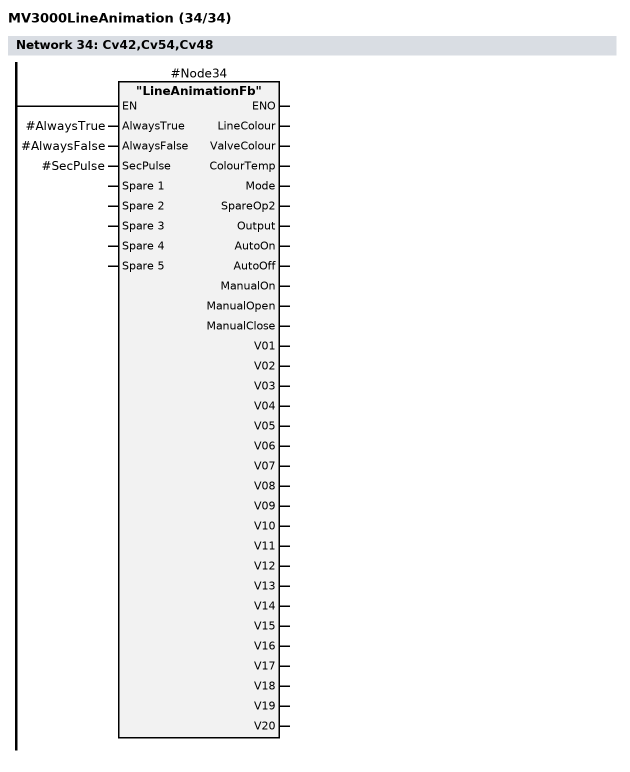
   RUNG wire#powerrail
      #Node34(AlwaysTrue := #AlwaysTrue, AlwaysFalse := #AlwaysFalse, SecPulse := #SecPulse, "Spare 1" :=, "Spare 2" :=, "Spare 3" :=, "Spare 4" :=, "Spare 5" :=, LineColour =>, ValveColour =>, ColourTemp =>, Mode =>, SpareOp2 =>, Output =>, AutoOn =>, AutoOff =>, ManualOn =>, ManualOpen =>, ManualClose =>, V01 =>, V02 =>, V03 =>, V04 =>, V05 =>, V06 =>, V07 =>, V08 =>, V09 =>, V10 =>, V11 =>, V12 =>, V13 =>, V14 =>, V15 =>, V16 =>, V17 =>, V18 =>, V19 =>, V20 =>)
   END_RUNG
   // the same network as SCL:
   #Node34(AlwaysTrue := #AlwaysTrue, AlwaysFalse := #AlwaysFalse, SecPulse := #SecPulse);   // "LineAnimationFb"
END_REGION
END_FUNCTION_BLOCK

FUNCTION_BLOCK "LineAnimationFb"   // FB802, LAD
{ S7_Optimized_Access := 'FALSE' }
// stored: AutoNumber false, SetENOAutomatically false
   VAR_INPUT
      AlwaysTrue : Bool;
      AlwaysFalse : Bool;
      SecPulse : Bool;
      "Spare 1" : Bool;
      "Spare 2" : Bool;
      "Spare 3" : Bool;
      "Spare 4" : Bool;
      "Spare 5" : Bool;
   END_VAR
   VAR_OUTPUT
      LineColour : DInt;
      ValveColour : DInt;
      ColourTemp : Int;
      Mode : Int;   // 0 - Force Close, 1- AutoOn, 2-ForceOn
      SpareOp2 : Int;
      Output : Bool;
      AutoOn : Bool;
      AutoOff : Bool;
      ManualOn : Bool;
      ManualOpen : Bool;
      ManualClose : Bool;
      V01 { ExternalAccessible := 'False'; ExternalVisible := 'False'; ExternalWritable := 'False'} : "LineAnimation";
      V02 { ExternalAccessible := 'False'; ExternalVisible := 'False'; ExternalWritable := 'False'} : "LineAnimation";
      V03 { ExternalAccessible := 'False'; ExternalVisible := 'False'; ExternalWritable := 'False'} : "LineAnimation";
      V04 { ExternalAccessible := 'False'; ExternalVisible := 'False'; ExternalWritable := 'False'} : "LineAnimation";
      V05 { ExternalAccessible := 'False'; ExternalVisible := 'False'; ExternalWritable := 'False'} : "LineAnimation";
      V06 { ExternalAccessible := 'False'; ExternalVisible := 'False'; ExternalWritable := 'False'} : "LineAnimation";
      V07 { ExternalAccessible := 'False'; ExternalVisible := 'False'; ExternalWritable := 'False'} : "LineAnimation";
      V08 { ExternalAccessible := 'False'; ExternalVisible := 'False'; ExternalWritable := 'False'} : "LineAnimation";
      V09 { ExternalAccessible := 'False'; ExternalVisible := 'False'; ExternalWritable := 'False'} : "LineAnimation";
      V10 { ExternalAccessible := 'False'; ExternalVisible := 'False'; ExternalWritable := 'False'} : "LineAnimation";
      V11 { ExternalAccessible := 'False'; ExternalVisible := 'False'; ExternalWritable := 'False'} : "LineAnimation";
      V12 { ExternalAccessible := 'False'; ExternalVisible := 'False'; ExternalWritable := 'False'} : "LineAnimation";
      V13 { ExternalAccessible := 'False'; ExternalVisible := 'False'; ExternalWritable := 'False'} : "LineAnimation";
      V14 { ExternalAccessible := 'False'; ExternalVisible := 'False'; ExternalWritable := 'False'} : "LineAnimation";
      V15 { ExternalAccessible := 'False'; ExternalVisible := 'False'; ExternalWritable := 'False'} : "LineAnimation";
      V16 { ExternalAccessible := 'False'; ExternalVisible := 'False'; ExternalWritable := 'False'} : "LineAnimation";
      V17 { ExternalAccessible := 'False'; ExternalVisible := 'False'; ExternalWritable := 'False'} : "LineAnimation";
      V18 { ExternalAccessible := 'False'; ExternalVisible := 'False'; ExternalWritable := 'False'} : "LineAnimation";
      V19 { ExternalAccessible := 'False'; ExternalVisible := 'False'; ExternalWritable := 'False'} : "LineAnimation";
      V20 { ExternalAccessible := 'False'; ExternalVisible := 'False'; ExternalWritable := 'False'} : "LineAnimation";
   END_VAR
BEGIN

REGION Network 1: Auto On
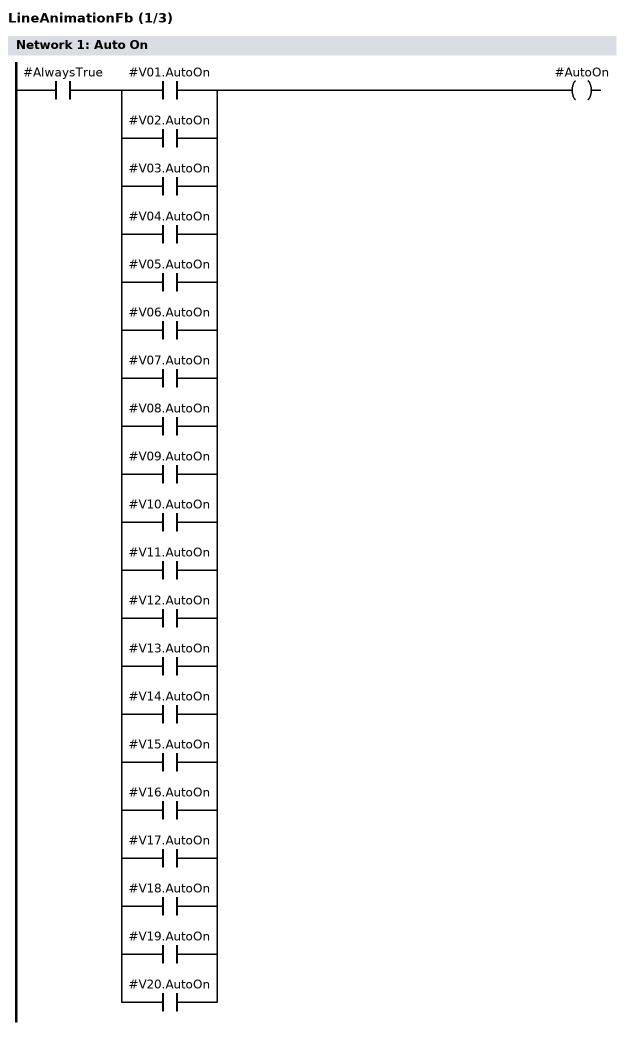
   RUNG wire#powerrail
      Contact( #AlwaysTrue )
      wire#w1
      Contact( #V01.AutoOn )
      wire#w2
      Coil( #AutoOn )
   END_RUNG
   RUNG wire#w1
      Contact( #V02.AutoOn )
   END_RUNG wire#w2
   RUNG wire#w1
      Contact( #V03.AutoOn )
   END_RUNG wire#w2
   RUNG wire#w1
      Contact( #V04.AutoOn )
   END_RUNG wire#w2
   RUNG wire#w1
      Contact( #V05.AutoOn )
   END_RUNG wire#w2
   RUNG wire#w1
      Contact( #V06.AutoOn )
   END_RUNG wire#w2
   RUNG wire#w1
      Contact( #V07.AutoOn )
   END_RUNG wire#w2
   RUNG wire#w1
      Contact( #V08.AutoOn )
   END_RUNG wire#w2
   RUNG wire#w1
      Contact( #V09.AutoOn )
   END_RUNG wire#w2
   RUNG wire#w1
      Contact( #V10.AutoOn )
   END_RUNG wire#w2
   RUNG wire#w1
      Contact( #V11.AutoOn )
   END_RUNG wire#w2
   RUNG wire#w1
      Contact( #V12.AutoOn )
   END_RUNG wire#w2
   RUNG wire#w1
      Contact( #V13.AutoOn )
   END_RUNG wire#w2
   RUNG wire#w1
      Contact( #V14.AutoOn )
   END_RUNG wire#w2
   RUNG wire#w1
      Contact( #V15.AutoOn )
   END_RUNG wire#w2
   RUNG wire#w1
      Contact( #V16.AutoOn )
   END_RUNG wire#w2
   RUNG wire#w1
      Contact( #V17.AutoOn )
   END_RUNG wire#w2
   RUNG wire#w1
      Contact( #V18.AutoOn )
   END_RUNG wire#w2
   RUNG wire#w1
      Contact( #V19.AutoOn )
   END_RUNG wire#w2
   RUNG wire#w1
      Contact( #V20.AutoOn )
   END_RUNG wire#w2
   // the same network as SCL:
   #AutoOn := #AlwaysTrue AND (#V01.AutoOn OR #V02.AutoOn OR #V03.AutoOn OR #V04.AutoOn OR #V05.AutoOn OR #V06.AutoOn OR #V07.AutoOn OR #V08.AutoOn OR #V09.AutoOn OR #V10.AutoOn OR #V11.AutoOn OR #V12.AutoOn OR #V13.AutoOn OR #V14.AutoOn OR #V15.AutoOn OR #V16.AutoOn OR #V17.AutoOn OR #V18.AutoOn OR #V19.AutoOn OR #V20.AutoOn);
END_REGION

REGION Network 2: Force Open
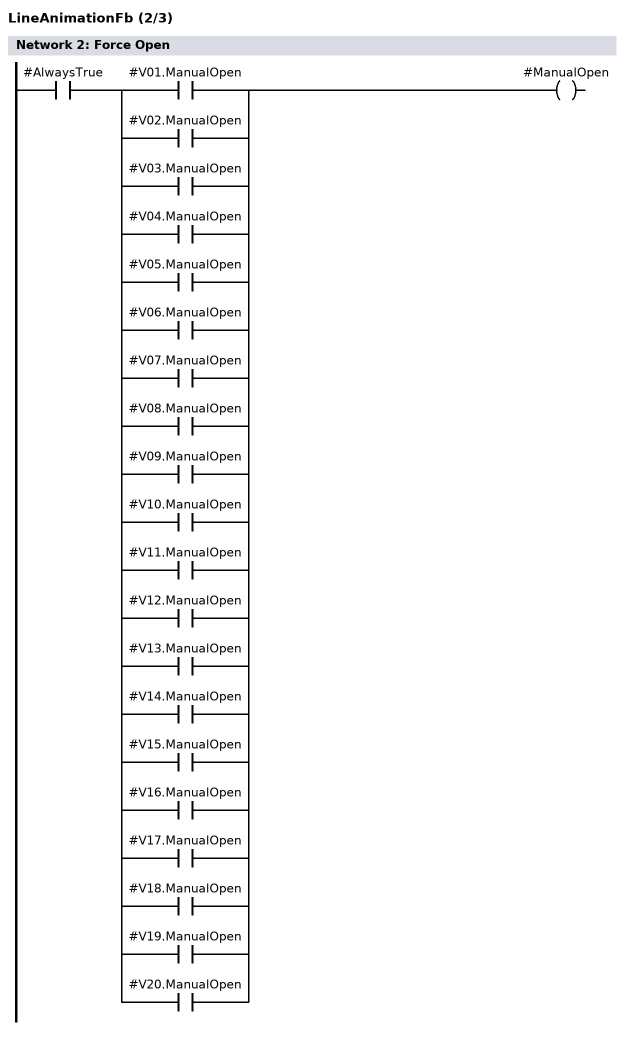
   RUNG wire#powerrail
      Contact( #AlwaysTrue )
      wire#w1
      Contact( #V01.ManualOpen )
      wire#w2
      Coil( #ManualOpen )
   END_RUNG
   RUNG wire#w1
      Contact( #V02.ManualOpen )
   END_RUNG wire#w2
   RUNG wire#w1
      Contact( #V03.ManualOpen )
   END_RUNG wire#w2
   RUNG wire#w1
      Contact( #V04.ManualOpen )
   END_RUNG wire#w2
   RUNG wire#w1
      Contact( #V05.ManualOpen )
   END_RUNG wire#w2
   RUNG wire#w1
      Contact( #V06.ManualOpen )
   END_RUNG wire#w2
   RUNG wire#w1
      Contact( #V07.ManualOpen )
   END_RUNG wire#w2
   RUNG wire#w1
      Contact( #V08.ManualOpen )
   END_RUNG wire#w2
   RUNG wire#w1
      Contact( #V09.ManualOpen )
   END_RUNG wire#w2
   RUNG wire#w1
      Contact( #V10.ManualOpen )
   END_RUNG wire#w2
   RUNG wire#w1
      Contact( #V11.ManualOpen )
   END_RUNG wire#w2
   RUNG wire#w1
      Contact( #V12.ManualOpen )
   END_RUNG wire#w2
   RUNG wire#w1
      Contact( #V13.ManualOpen )
   END_RUNG wire#w2
   RUNG wire#w1
      Contact( #V14.ManualOpen )
   END_RUNG wire#w2
   RUNG wire#w1
      Contact( #V15.ManualOpen )
   END_RUNG wire#w2
   RUNG wire#w1
      Contact( #V16.ManualOpen )
   END_RUNG wire#w2
   RUNG wire#w1
      Contact( #V17.ManualOpen )
   END_RUNG wire#w2
   RUNG wire#w1
      Contact( #V18.ManualOpen )
   END_RUNG wire#w2
   RUNG wire#w1
      Contact( #V19.ManualOpen )
   END_RUNG wire#w2
   RUNG wire#w1
      Contact( #V20.ManualOpen )
   END_RUNG wire#w2
   // the same network as SCL:
   #ManualOpen := #AlwaysTrue AND (#V01.ManualOpen OR #V02.ManualOpen OR #V03.ManualOpen OR #V04.ManualOpen OR #V05.ManualOpen OR #V06.ManualOpen OR #V07.ManualOpen OR #V08.ManualOpen OR #V09.ManualOpen OR #V10.ManualOpen OR #V11.ManualOpen OR #V12.ManualOpen OR #V13.ManualOpen OR #V14.ManualOpen OR #V15.ManualOpen OR #V16.ManualOpen OR #V17.ManualOpen OR #V18.ManualOpen OR #V19.ManualOpen OR #V20.ManualOpen);
END_REGION

REGION Network 3: Line Colour
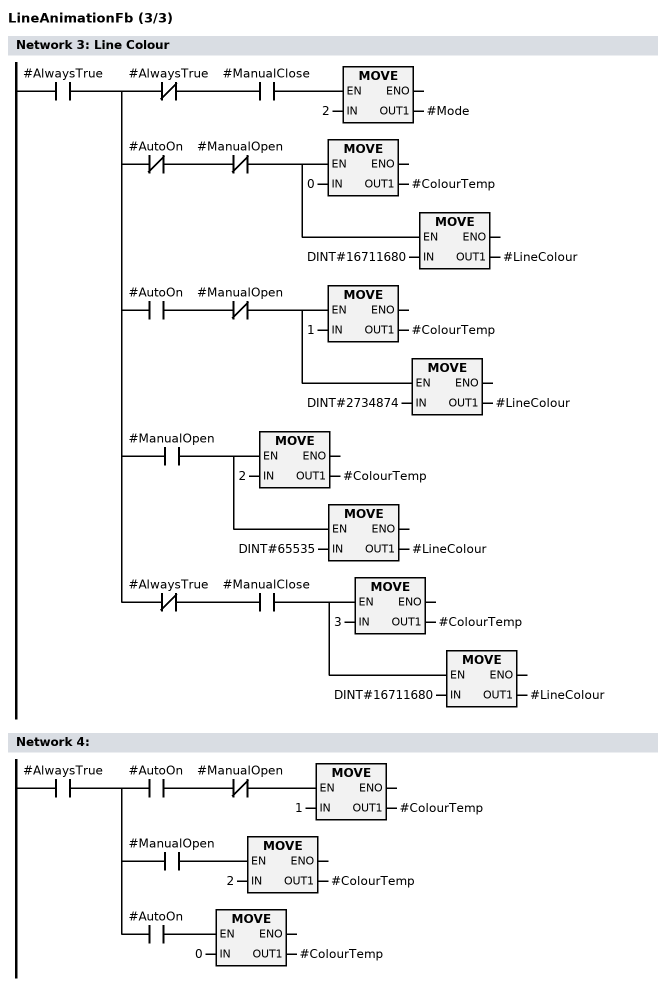
   RUNG wire#powerrail
      Contact( #AlwaysTrue )
      wire#w1
      I_Contact( #AlwaysTrue )
      Contact( #ManualClose )
      Move(in := 2, out1 => #Mode)
   END_RUNG
   RUNG wire#w1
      I_Contact( #AutoOn )
      I_Contact( #ManualOpen )
      wire#w2
      Move(in := 0, out1 => #ColourTemp)
   END_RUNG
   RUNG wire#w2
      Move(in := DINT#16711680, out1 => #LineColour)
   END_RUNG
   RUNG wire#w1
      Contact( #AutoOn )
      I_Contact( #ManualOpen )
      wire#w3
      Move(in := 1, out1 => #ColourTemp)
   END_RUNG
   RUNG wire#w3
      Move(in := DINT#2734874, out1 => #LineColour)
   END_RUNG
   RUNG wire#w1
      Contact( #ManualOpen )
      wire#w4
      Move(in := 2, out1 => #ColourTemp)
   END_RUNG
   RUNG wire#w4
      Move(in := DINT#65535, out1 => #LineColour)
   END_RUNG
   RUNG wire#w1
      I_Contact( #AlwaysTrue )
      Contact( #ManualClose )
      wire#w5
      Move(in := 3, out1 => #ColourTemp)
   END_RUNG
   RUNG wire#w5
      Move(in := DINT#16711680, out1 => #LineColour)
   END_RUNG
   // the same network as SCL:
   IF #AlwaysTrue AND NOT #AlwaysTrue AND #ManualClose THEN #Mode := 2; END_IF;
   IF #AlwaysTrue AND NOT #AutoOn AND NOT #ManualOpen THEN
       #ColourTemp := 0;
       #LineColour := DINT#16711680;
   END_IF;
   IF #AlwaysTrue AND #AutoOn AND NOT #ManualOpen THEN
       #ColourTemp := 1;
       #LineColour := DINT#2734874;
   END_IF;
   IF #AlwaysTrue AND #ManualOpen THEN
       #ColourTemp := 2;
       #LineColour := DINT#65535;
   END_IF;
   IF #AlwaysTrue AND NOT #AlwaysTrue AND #ManualClose THEN
       #ColourTemp := 3;
       #LineColour := DINT#16711680;
   END_IF;
END_REGION

REGION Network 4
   RUNG wire#powerrail
      Contact( #AlwaysTrue )
      wire#w1
      Contact( #AutoOn )
      I_Contact( #ManualOpen )
      Move(in := 1, out1 => #ColourTemp)
   END_RUNG
   RUNG wire#w1
      Contact( #ManualOpen )
      Move(in := 2, out1 => #ColourTemp)
   END_RUNG
   RUNG wire#w1
      Contact( #AutoOn )
      Move(in := 0, out1 => #ColourTemp)
   END_RUNG
   // the same network as SCL:
   IF #AlwaysTrue AND #AutoOn AND NOT #ManualOpen THEN #ColourTemp := 1; END_IF;
   IF #AlwaysTrue AND #ManualOpen THEN #ColourTemp := 2; END_IF;
   IF #AlwaysTrue AND #AutoOn THEN #ColourTemp := 0; END_IF;
END_REGION
END_FUNCTION_BLOCK

FUNCTION "MV3000LineAnimationFc" : Void
{ S7_Optimized_Access := 'FALSE' }
VERSION : 0.1

BEGIN
	//////////////////////////////////// AUTO ON ////////////////////////////////////////////
	//AutoON
	"MV3000LineAnimationDb"."Node 1".V01.AutoOn := "ValvesOutputDb".Cv01;
	"MV3000LineAnimationDb"."Node 1".V02.AutoOn := "ValvesOutputDb".Cv02;
	"MV3000LineAnimationDb"."Node 1".V03.AutoOn := "ValvesOutputDb".Cv10;
	
	
	"MV3000LineAnimationDb"."Node 2".V01.AutoOn := "ValvesOutputDb".Cv03;
	"MV3000LineAnimationDb"."Node 2".V02.AutoOn := "ValvesOutputDb".Cv04;
	"MV3000LineAnimationDb"."Node 2".V03.AutoOn := "ValvesOutputDb".Cv05;
	"MV3000LineAnimationDb"."Node 2".V04.AutoOn := "ValvesOutputDb".Cv06;
	
	
	"MV3000LineAnimationDb"."Node 3".V01.AutoOn := "ValvesOutputDb".Cv07;
	"MV3000LineAnimationDb"."Node 3".V02.AutoOn := "ValvesOutputDb".Cv08;
	"MV3000LineAnimationDb"."Node 3".V03.AutoOn := "ValvesOutputDb".Cv09;
	
	
	"MV3000LineAnimationDb"."Node 4".V01.AutoOn := "ValvesOutputDb".Cv16;
	"MV3000LineAnimationDb"."Node 4".V02.AutoOn := "ValvesOutputDb".Cv17;
	"MV3000LineAnimationDb"."Node 4".V03.AutoOn := "ValvesOutputDb".Cv22;
	"MV3000LineAnimationDb"."Node 4".V04.AutoOn := "ValvesOutputDb".Cv23;
	"MV3000LineAnimationDb"."Node 4".V05.AutoOn := "ValvesOutputDb".Cv24;
	"MV3000LineAnimationDb"."Node 4".V06.AutoOn := "ValvesOutputDb".Cv25;
	
	
	"MV3000LineAnimationDb"."Node 5".V01.AutoOn := "ValvesOutputDb".Cv22;
	"MV3000LineAnimationDb"."Node 5".V02.AutoOn := "ValvesOutputDb".Cv25;
	
	
	"MV3000LineAnimationDb"."Node 6".V01.AutoOn := "ValvesOutputDb".Cv18;
	"MV3000LineAnimationDb"."Node 6".V02.AutoOn := "ValvesOutputDb".Cv19;
	"MV3000LineAnimationDb"."Node 6".V03.AutoOn := "ValvesOutputDb".Cv20;
	"MV3000LineAnimationDb"."Node 6".V04.AutoOn := "ValvesOutputDb".Cv21;
	
	"MV3000LineAnimationDb"."Node 7".V01.AutoOn := "ValvesOutputDb".Cv19;
	"MV3000LineAnimationDb"."Node 7".V02.AutoOn := "ValvesOutputDb".Cv20;
	
	"MV3000LineAnimationDb"."Node 8".V01.AutoOn := "ValvesOutputDb".Cv16;
	"MV3000LineAnimationDb"."Node 8".V02.AutoOn := "ValvesOutputDb".Cv15;
	"MV3000LineAnimationDb"."Node 8".V03.AutoOn := "ValvesOutputDb".Cv63;
	
	"MV3000LineAnimationDb"."Node 9".V01.AutoOn := "ValvesOutputDb".Cv10;
	"MV3000LineAnimationDb"."Node 9".V02.AutoOn := "ValvesOutputDb".Cv11;
	"MV3000LineAnimationDb"."Node 9".V03.AutoOn := "ValvesOutputDb".Cv12;
	"MV3000LineAnimationDb"."Node 9".V04.AutoOn := "ValvesOutputDb".Cv13;
	"MV3000LineAnimationDb"."Node 9".V05.AutoOn := "ValvesOutputDb".Cv14;
	"MV3000LineAnimationDb"."Node 9".V06.AutoOn := "ValvesOutputDb".Cv15;
	
	"MV3000LineAnimationDb"."Node 10".V01.AutoOn := "ValvesOutputDb".Cv11;
	"MV3000LineAnimationDb"."Node 10".V02.AutoOn := "ValvesOutputDb".Cv39;
	
	"MV3000LineAnimationDb"."Node 11".V01.AutoOn := "ValvesOutputDb".Cv12;
	"MV3000LineAnimationDb"."Node 11".V02.AutoOn := "ValvesOutputDb".Cv26;
	"MV3000LineAnimationDb"."Node 11".V03.AutoOn := "ValvesOutputDb".Cv64;
	
	"MV3000LineAnimationDb"."Node 12".V01.AutoOn := "ValvesOutputDb".Cv31;
	"MV3000LineAnimationDb"."Node 12".V02.AutoOn := "ValvesOutputDb".Cv41;
	
	"MV3000LineAnimationDb"."Node 13".V01.AutoOn := "ValvesOutputDb".Fbov01;
	"MV3000LineAnimationDb"."Node 13".V02.AutoOn := "ValvesOutputDb".Cv30;
	"MV3000LineAnimationDb"."Node 13".V03.AutoOn := "ValvesOutputDb".Cv31;
	"MV3000LineAnimationDb"."Node 13".V04.AutoOn := "ValvesOutputDb".Cv32;
	"MV3000LineAnimationDb"."Node 13".V05.AutoOn := "ValvesOutputDb".Cv33;
	
	"MV3000LineAnimationDb"."Node 14".V01.AutoOn := "ValvesOutputDb".Cv27;
	"MV3000LineAnimationDb"."Node 14".V02.AutoOn := "ValvesOutputDb".Cv28;
	"MV3000LineAnimationDb"."Node 14".V03.AutoOn := "ValvesOutputDb".Cv29;
	
	"MV3000LineAnimationDb"."Node 15".V01.AutoOn := "ValvesOutputDb".Cv30;
	"MV3000LineAnimationDb"."Node 15".V02.AutoOn := "ValvesOutputDb".Cv33;
	"MV3000LineAnimationDb"."Node 15".V03.AutoOn := "ValvesOutputDb".Cv34;
	"MV3000LineAnimationDb"."Node 15".V04.AutoOn := "ValvesOutputDb".Cv35;
	
	"MV3000LineAnimationDb"."Node 16".V01.AutoOn := "ValvesOutputDb".Cv32;
	"MV3000LineAnimationDb"."Node 16".V02.AutoOn := "ValvesOutputDb".Cv36;
	"MV3000LineAnimationDb"."Node 16".V03.AutoOn := "ValvesOutputDb".Cv39;
	"MV3000LineAnimationDb"."Node 16".V04.AutoOn := "ValvesOutputDb".Cv40;
	
	"MV3000LineAnimationDb"."Node 17".V01.AutoOn := "ValvesOutputDb".Cv40;
	"MV3000LineAnimationDb"."Node 17".V02.AutoOn := "ValvesOutputDb".Cv41;
	"MV3000LineAnimationDb"."Node 17".V03.AutoOn := "ValvesOutputDb".Cv42;
	"MV3000LineAnimationDb"."Node 17".V04.AutoOn := "ValvesOutputDb".Cv43;
	"MV3000LineAnimationDb"."Node 17".V05.AutoOn := "ValvesOutputDb".Cv44;
	
	"MV3000LineAnimationDb"."Node 18".V01.AutoOn := "ValvesOutputDb".Cv43;
	"MV3000LineAnimationDb"."Node 18".V02.AutoOn := "ValvesOutputDb".Cv47;
	"MV3000LineAnimationDb"."Node 18".V03.AutoOn := "ValvesOutputDb".Cv48;
	"MV3000LineAnimationDb"."Node 18".V04.AutoOn := "ValvesOutputDb".Cv49;
	"MV3000LineAnimationDb"."Node 18".V05.AutoOn := "ValvesOutputDb".Cv50;
	
	
	"MV3000LineAnimationDb"."Node 19".V01.AutoOn := "ValvesOutputDb".Cv49;
	"MV3000LineAnimationDb"."Node 19".V02.AutoOn := "ValvesOutputDb".Cv53;
	"MV3000LineAnimationDb"."Node 19".V03.AutoOn := "ValvesOutputDb".Cv54;
	"MV3000LineAnimationDb"."Node 19".V04.AutoOn := "ValvesOutputDb".Cv55;
	"MV3000LineAnimationDb"."Node 19".V05.AutoOn := "ValvesOutputDb".Cv56;
	
	"MV3000LineAnimationDb"."Node 20".V01.AutoOn := "ValvesOutputDb".Cv55;
	"MV3000LineAnimationDb"."Node 20".V02.AutoOn := "ValvesOutputDb".Cv61;
	"MV3000LineAnimationDb"."Node 20".V03.AutoOn := "ValvesOutputDb".Cv62;
	
	
	"MV3000LineAnimationDb"."Node 21".V01.AutoOn := "ValvesOutputDb".Cv59;
	"MV3000LineAnimationDb"."Node 21".V02.AutoOn := "ValvesOutputDb".Cv60;
	"MV3000LineAnimationDb"."Node 21".V03.AutoOn := "ValvesOutputDb".Cv61;
	
	"MV3000LineAnimationDb"."Node 22".V01.AutoOn := "ValvesOutputDb".Cv56;
	"MV3000LineAnimationDb"."Node 22".V02.AutoOn := "ValvesOutputDb".Cv58;
	"MV3000LineAnimationDb"."Node 22".V03.AutoOn := "ValvesOutputDb".Cv57;
	
	"MV3000LineAnimationDb"."Node 23".V01.AutoOn := "ValvesOutputDb".Cv50;
	"MV3000LineAnimationDb"."Node 23".V02.AutoOn := "ValvesOutputDb".Cv51;
	"MV3000LineAnimationDb"."Node 23".V03.AutoOn := "ValvesOutputDb".Cv52;
	"MV3000LineAnimationDb"."Node 23".V04.AutoOn := "ValvesOutputDb".Cv53;
	
	
	"MV3000LineAnimationDb"."Node 24".V01.AutoOn := "ValvesOutputDb".Cv44;
	"MV3000LineAnimationDb"."Node 24".V02.AutoOn := "ValvesOutputDb".Cv45;
	"MV3000LineAnimationDb"."Node 24".V03.AutoOn := "ValvesOutputDb".Cv46;
	"MV3000LineAnimationDb"."Node 24".V04.AutoOn := "ValvesOutputDb".Cv47;
	
	"MV3000LineAnimationDb"."Node 25".V01.AutoOn := "ValvesOutputDb".Cv36;
	"MV3000LineAnimationDb"."Node 25".V02.AutoOn := "ValvesOutputDb".Cv37;
	"MV3000LineAnimationDb"."Node 25".V03.AutoOn := "ValvesOutputDb".Cv38;
	
	
	"MV3000LineAnimationDb"."Node 26".V01.AutoOn := "ValvesOutputDb".Cv30;
	"MV3000LineAnimationDb"."Node 26".V02.AutoOn := "ValvesOutputDb".Cv33;
	"MV3000LineAnimationDb"."Node 26".V03.AutoOn := "ValvesOutputDb".Cv34;
	"MV3000LineAnimationDb"."Node 26".V04.AutoOn := "ValvesOutputDb".Cv35;
	
	"MV3000LineAnimationDb"."Node 27".V01.AutoOn := "ValvesOutputDb".Cv28;
	"MV3000LineAnimationDb"."Node 27".V02.AutoOn := "ValvesOutputDb".Cv34;
	"MV3000LineAnimationDb"."Node 27".V03.AutoOn := "ValvesOutputDb".Cv37;
	"MV3000LineAnimationDb"."Node 27".V04.AutoOn := "ValvesOutputDb".Cv45;
	"MV3000LineAnimationDb"."Node 27".V05.AutoOn := "ValvesOutputDb".Cv51;
	"MV3000LineAnimationDb"."Node 27".V06.AutoOn := "ValvesOutputDb".Cv57;
	"MV3000LineAnimationDb"."Node 27".V07.AutoOn := "ValvesOutputDb".Cv60;
	
	"MV3000LineAnimationDb"."Node 28".V01.AutoOn := "ValvesOutputDb".Cv22;
	"MV3000LineAnimationDb"."Node 28".V02.AutoOn := "ValvesOutputDb".Cv19;
	"MV3000LineAnimationDb"."Node 28".V03.AutoOn := "ValvesOutputDb".Cv25;
	"MV3000LineAnimationDb"."Node 28".V04.AutoOn := "ValvesOutputDb".Cv20;
	"MV3000LineAnimationDb"."Node 28".V05.AutoOn := "ValvesOutputDb".Cv29;
	"MV3000LineAnimationDb"."Node 28".V06.AutoOn := "ValvesOutputDb".Cv35;
	"MV3000LineAnimationDb"."Node 28".V07.AutoOn := "ValvesOutputDb".Cv38;
	"MV3000LineAnimationDb"."Node 28".V08.AutoOn := "ValvesOutputDb".Cv46;
	"MV3000LineAnimationDb"."Node 28".V09.AutoOn := "ValvesOutputDb".Cv52;
	"MV3000LineAnimationDb"."Node 28".V10.AutoOn := "ValvesOutputDb".Cv58;
	"MV3000LineAnimationDb"."Node 28".V11.AutoOn := "ValvesOutputDb".Cv59;
	
	"MV3000LineAnimationDb"."Node 29".V01.AutoOn := "ValvesOutputDb".Cv04;
	"MV3000LineAnimationDb"."Node 29".V02.AutoOn := "ValvesOutputDb".Cv01;
	
	"MV3000LineAnimationDb"."Node 30".V01.AutoOn := "ValvesOutputDb".Cv06;
	"MV3000LineAnimationDb"."Node 30".V02.AutoOn := "ValvesOutputDb".Cv09;
	
	"MV3000LineAnimationDb"."Node31".V01.AutoOn :="ValvesOutputDb".Cv06;
	"MV3000LineAnimationDb"."Node31".V02.AutoOn := "ValvesOutputDb".Cv09;
	"MV3000LineAnimationDb"."Node31".V03.AutoOn := "ValvesOutputDb".Cv08;
	
	"MV3000LineAnimationDb".Node32.V01.AutoOn := "ValvesOutputDb".Cv05;
	"MV3000LineAnimationDb".Node32.V02.AutoOn := "ValvesOutputDb".Cv24;
	
	"MV3000LineAnimationDb".Node33.V01.AutoOn := "ValvesOutputDb".Fbov01;
	"MV3000LineAnimationDb".Node33.V02.AutoOn := "ValvesOutputDb".Cv26;
	
	
	"MV3000LineAnimationDb".Node34.V01.AutoOn := "ValvesOutputDb".Cv42;
	"MV3000LineAnimationDb".Node34.V02.AutoOn := "ValvesOutputDb".Cv54;
	"MV3000LineAnimationDb".Node34.V03.AutoOn := "ValvesOutputDb".Cv48;
	
	
	
	
	
	//////////////////////////////////////////  MANUAL OPEN /////////////////////////////////////////////
	
	//ManualOpen
	
	"MV3000LineAnimationDb"."Node 1".V01.ManualOpen := "DO_FaceplateDb".Cv01.ValveOpen;
	"MV3000LineAnimationDb"."Node 1".V02.ManualOpen := "DO_FaceplateDb".Cv02.ValveOpen;
	"MV3000LineAnimationDb"."Node 1".V03.ManualOpen := "DO_FaceplateDb".Cv10.ValveOpen;
	
	
	"MV3000LineAnimationDb"."Node 2".V01.ManualOpen := "DO_FaceplateDb".Cv03.ValveOpen;
	"MV3000LineAnimationDb"."Node 2".V02.ManualOpen := "DO_FaceplateDb".Cv04.ValveOpen;
	"MV3000LineAnimationDb"."Node 2".V03.ManualOpen := "DO_FaceplateDb".Cv05.ValveOpen;
	"MV3000LineAnimationDb"."Node 2".V04.ManualOpen := "DO_FaceplateDb".Cv06.ValveOpen;
	
	
	"MV3000LineAnimationDb"."Node 3".V01.ManualOpen := "DO_FaceplateDb".Cv07.ValveOpen;
	"MV3000LineAnimationDb"."Node 3".V02.ManualOpen := "DO_FaceplateDb".Cv08.ValveOpen;
	"MV3000LineAnimationDb"."Node 3".V03.ManualOpen := "DO_FaceplateDb".Cv09.ValveOpen;
	
	
	"MV3000LineAnimationDb"."Node 4".V01.ManualOpen := "DO_FaceplateDb".Cv16.ValveOpen;
	"MV3000LineAnimationDb"."Node 4".V02.ManualOpen := "DO_FaceplateDb".Cv17.ValveOpen;
	"MV3000LineAnimationDb"."Node 4".V03.ManualOpen := "DO_FaceplateDb".Cv22.ValveOpen;
	"MV3000LineAnimationDb"."Node 4".V04.ManualOpen := "DO_FaceplateDb".Cv23.ValveOpen;
	"MV3000LineAnimationDb"."Node 4".V05.ManualOpen := "DO_FaceplateDb".Cv24.ValveOpen;
	"MV3000LineAnimationDb"."Node 4".V06.ManualOpen := "DO_FaceplateDb".Cv25.ValveOpen;
	
	
	"MV3000LineAnimationDb"."Node 5".V01.ManualOpen := "DO_FaceplateDb".Cv22.ValveOpen;
	"MV3000LineAnimationDb"."Node 5".V02.ManualOpen := "DO_FaceplateDb".Cv25.ValveOpen;
	
	
	"MV3000LineAnimationDb"."Node 6".V01.ManualOpen := "DO_FaceplateDb".Cv18.ValveOpen;
	"MV3000LineAnimationDb"."Node 6".V02.ManualOpen := "DO_FaceplateDb".Cv19.ValveOpen;
	"MV3000LineAnimationDb"."Node 6".V03.ManualOpen := "DO_FaceplateDb".Cv20.ValveOpen;
	"MV3000LineAnimationDb"."Node 6".V04.ManualOpen := "DO_FaceplateDb".Cv21.ValveOpen;
	
	"MV3000LineAnimationDb"."Node 7".V01.ManualOpen := "DO_FaceplateDb".Cv19.ValveOpen;
	"MV3000LineAnimationDb"."Node 7".V02.ManualOpen := "DO_FaceplateDb".Cv20.ValveOpen;
	
	"MV3000LineAnimationDb"."Node 8".V01.ManualOpen := "DO_FaceplateDb".Cv16.ValveOpen;
	"MV3000LineAnimationDb"."Node 8".V02.ManualOpen := "DO_FaceplateDb".Cv15.ValveOpen;
	"MV3000LineAnimationDb"."Node 8".V03.ManualOpen := "DO_FaceplateDb".Cv63.ValveOpen;
	
	"MV3000LineAnimationDb"."Node 9".V01.ManualOpen := "DO_FaceplateDb".Cv10.ValveOpen;
	"MV3000LineAnimationDb"."Node 9".V02.ManualOpen := "DO_FaceplateDb".Cv11.ValveOpen;
	"MV3000LineAnimationDb"."Node 9".V03.ManualOpen := "DO_FaceplateDb".Cv12.ValveOpen;
	"MV3000LineAnimationDb"."Node 9".V04.ManualOpen := "DO_FaceplateDb".Cv13.ValveOpen;
	"MV3000LineAnimationDb"."Node 9".V05.ManualOpen := "DO_FaceplateDb".Cv14.ValveOpen;
	"MV3000LineAnimationDb"."Node 9".V06.ManualOpen := "DO_FaceplateDb".Cv15.ValveOpen;
	
	"MV3000LineAnimationDb"."Node 10".V01.ManualOpen := "DO_FaceplateDb".Cv11.ValveOpen;
	"MV3000LineAnimationDb"."Node 10".V02.ManualOpen := "DO_FaceplateDb".Cv39.ValveOpen;
	
	"MV3000LineAnimationDb"."Node 11".V01.ManualOpen := "DO_FaceplateDb".Cv12.ValveOpen;
	"MV3000LineAnimationDb"."Node 11".V02.ManualOpen := "DO_FaceplateDb".Cv26.ValveOpen;
	"MV3000LineAnimationDb"."Node 11".V03.ManualOpen := "DO_FaceplateDb".Cv64.ValveOpen;
	
	"MV3000LineAnimationDb"."Node 12".V01.ManualOpen := "DO_FaceplateDb".Cv31.ValveOpen;
	"MV3000LineAnimationDb"."Node 12".V02.ManualOpen := "DO_FaceplateDb".Cv41.ValveOpen;
	
	"MV3000LineAnimationDb"."Node 13".V01.ManualOpen := "DO_FaceplateDb".Fbov01.ValveOpen;
	"MV3000LineAnimationDb"."Node 13".V02.ManualOpen := "DO_FaceplateDb".Cv30.ValveOpen;
	"MV3000LineAnimationDb"."Node 13".V03.ManualOpen := "DO_FaceplateDb".Cv31.ValveOpen;
	"MV3000LineAnimationDb"."Node 13".V04.ManualOpen := "DO_FaceplateDb".Cv32.ValveOpen;
	"MV3000LineAnimationDb"."Node 13".V05.ManualOpen := "DO_FaceplateDb".Cv33.ValveOpen;
	
	"MV3000LineAnimationDb"."Node 14".V01.ManualOpen := "DO_FaceplateDb".Cv27.ValveOpen;
	"MV3000LineAnimationDb"."Node 14".V02.ManualOpen := "DO_FaceplateDb".Cv28.ValveOpen;
	"MV3000LineAnimationDb"."Node 14".V03.ManualOpen := "DO_FaceplateDb".Cv29.ValveOpen;
	
	"MV3000LineAnimationDb"."Node 15".V01.ManualOpen := "DO_FaceplateDb".Cv30.ValveOpen;
	"MV3000LineAnimationDb"."Node 15".V02.ManualOpen := "DO_FaceplateDb".Cv33.ValveOpen;
	"MV3000LineAnimationDb"."Node 15".V03.ManualOpen := "DO_FaceplateDb".Cv34.ValveOpen;
	"MV3000LineAnimationDb"."Node 15".V04.ManualOpen := "DO_FaceplateDb".Cv35.ValveOpen;
	
	"MV3000LineAnimationDb"."Node 16".V01.ManualOpen := "DO_FaceplateDb".Cv32.ValveOpen;
	"MV3000LineAnimationDb"."Node 16".V02.ManualOpen := "DO_FaceplateDb".Cv36.ValveOpen;
	"MV3000LineAnimationDb"."Node 16".V03.ManualOpen := "DO_FaceplateDb".Cv39.ValveOpen;
	"MV3000LineAnimationDb"."Node 16".V04.ManualOpen := "DO_FaceplateDb".Cv40.ValveOpen;
	
	"MV3000LineAnimationDb"."Node 17".V01.ManualOpen := "DO_FaceplateDb".Cv40.ValveOpen;
	"MV3000LineAnimationDb"."Node 17".V02.ManualOpen := "DO_FaceplateDb".Cv41.ValveOpen;
	"MV3000LineAnimationDb"."Node 17".V03.ManualOpen := "DO_FaceplateDb".Cv42.ValveOpen;
	"MV3000LineAnimationDb"."Node 17".V04.ManualOpen := "DO_FaceplateDb".Cv43.ValveOpen;
	"MV3000LineAnimationDb"."Node 17".V05.ManualOpen := "DO_FaceplateDb".Cv44.ValveOpen;
	
	"MV3000LineAnimationDb"."Node 18".V01.ManualOpen := "DO_FaceplateDb".Cv43.ValveOpen;
	"MV3000LineAnimationDb"."Node 18".V02.ManualOpen := "DO_FaceplateDb".Cv47.ValveOpen;
	"MV3000LineAnimationDb"."Node 18".V03.ManualOpen := "DO_FaceplateDb".Cv48.ValveOpen;
	"MV3000LineAnimationDb"."Node 18".V04.ManualOpen := "DO_FaceplateDb".Cv49.ValveOpen;
	"MV3000LineAnimationDb"."Node 18".V05.ManualOpen := "DO_FaceplateDb".Cv50.ValveOpen;
	
	
	"MV3000LineAnimationDb"."Node 19".V01.ManualOpen := "DO_FaceplateDb".Cv49.ValveOpen;
	"MV3000LineAnimationDb"."Node 19".V02.ManualOpen := "DO_FaceplateDb".Cv53.ValveOpen;
	"MV3000LineAnimationDb"."Node 19".V03.ManualOpen := "DO_FaceplateDb".Cv54.ValveOpen;
	"MV3000LineAnimationDb"."Node 19".V04.ManualOpen := "DO_FaceplateDb".Cv55.ValveOpen;
	"MV3000LineAnimationDb"."Node 19".V05.ManualOpen := "DO_FaceplateDb".Cv56.ValveOpen;
	
	"MV3000LineAnimationDb"."Node 20".V01.ManualOpen := "DO_FaceplateDb".Cv55.ValveOpen;
	"MV3000LineAnimationDb"."Node 20".V02.ManualOpen := "DO_FaceplateDb".Cv61.ValveOpen;
	"MV3000LineAnimationDb"."Node 20".V03.ManualOpen := "DO_FaceplateDb".Cv62.ValveOpen;
	
	
	"MV3000LineAnimationDb"."Node 21".V01.ManualOpen := "DO_FaceplateDb".Cv59.ValveOpen;
	"MV3000LineAnimationDb"."Node 21".V02.ManualOpen := "DO_FaceplateDb".Cv60.ValveOpen;
	"MV3000LineAnimationDb"."Node 21".V03.ManualOpen := "DO_FaceplateDb".Cv61.ValveOpen;
	
	"MV3000LineAnimationDb"."Node 22".V01.ManualOpen := "DO_FaceplateDb".Cv56.ValveOpen;
	"MV3000LineAnimationDb"."Node 22".V02.ManualOpen := "DO_FaceplateDb".Cv58.ValveOpen;
	"MV3000LineAnimationDb"."Node 22".V03.ManualOpen := "DO_FaceplateDb".Cv57.ValveOpen;
	
	"MV3000LineAnimationDb"."Node 23".V01.ManualOpen := "DO_FaceplateDb".Cv50.ValveOpen;
	"MV3000LineAnimationDb"."Node 23".V02.ManualOpen := "DO_FaceplateDb".Cv51.ValveOpen;
	"MV3000LineAnimationDb"."Node 23".V03.ManualOpen := "DO_FaceplateDb".Cv52.ValveOpen;
	"MV3000LineAnimationDb"."Node 23".V04.ManualOpen := "DO_FaceplateDb".Cv53.ValveOpen;
	
	
	"MV3000LineAnimationDb"."Node 24".V01.ManualOpen := "DO_FaceplateDb".Cv44.ValveOpen;
	"MV3000LineAnimationDb"."Node 24".V02.ManualOpen := "DO_FaceplateDb".Cv45.ValveOpen;
	"MV3000LineAnimationDb"."Node 24".V03.ManualOpen := "DO_FaceplateDb".Cv46.ValveOpen;
	"MV3000LineAnimationDb"."Node 24".V04.ManualOpen := "DO_FaceplateDb".Cv47.ValveOpen;
	
	"MV3000LineAnimationDb"."Node 25".V01.ManualOpen := "DO_FaceplateDb".Cv36.ValveOpen;
	"MV3000LineAnimationDb"."Node 25".V02.ManualOpen := "DO_FaceplateDb".Cv37.ValveOpen;
	"MV3000LineAnimationDb"."Node 25".V03.ManualOpen := "DO_FaceplateDb".Cv38.ValveOpen;
	
	
	"MV3000LineAnimationDb"."Node 26".V01.ManualOpen := "DO_FaceplateDb".Cv30.ValveOpen;
	"MV3000LineAnimationDb"."Node 26".V02.ManualOpen := "DO_FaceplateDb".Cv33.ValveOpen;
	"MV3000LineAnimationDb"."Node 26".V03.ManualOpen := "DO_FaceplateDb".Cv34.ValveOpen;
	"MV3000LineAnimationDb"."Node 26".V04.ManualOpen := "DO_FaceplateDb".Cv35.ValveOpen;
	
	"MV3000LineAnimationDb"."Node 27".V01.ManualOpen := "DO_FaceplateDb".Cv28.ValveOpen;
	"MV3000LineAnimationDb"."Node 27".V02.ManualOpen := "DO_FaceplateDb".Cv34.ValveOpen;
	"MV3000LineAnimationDb"."Node 27".V03.ManualOpen := "DO_FaceplateDb".Cv37.ValveOpen;
	"MV3000LineAnimationDb"."Node 27".V04.ManualOpen := "DO_FaceplateDb".Cv45.ValveOpen;
	"MV3000LineAnimationDb"."Node 27".V05.ManualOpen := "DO_FaceplateDb".Cv51.ValveOpen;
	"MV3000LineAnimationDb"."Node 27".V06.ManualOpen := "DO_FaceplateDb".Cv57.ValveOpen;
	"MV3000LineAnimationDb"."Node 27".V07.ManualOpen := "DO_FaceplateDb".Cv60.ValveOpen;
	
	"MV3000LineAnimationDb"."Node 28".V01.ManualOpen := "DO_FaceplateDb".Cv22.ValveOpen;
	"MV3000LineAnimationDb"."Node 28".V02.ManualOpen := "DO_FaceplateDb".Cv19.ValveOpen;
	"MV3000LineAnimationDb"."Node 28".V03.ManualOpen := "DO_FaceplateDb".Cv25.ValveOpen;
	"MV3000LineAnimationDb"."Node 28".V04.ManualOpen := "DO_FaceplateDb".Cv20.ValveOpen;
	"MV3000LineAnimationDb"."Node 28".V05.ManualOpen := "DO_FaceplateDb".Cv29.ValveOpen;
	"MV3000LineAnimationDb"."Node 28".V06.ManualOpen := "DO_FaceplateDb".Cv35.ValveOpen;
	"MV3000LineAnimationDb"."Node 28".V07.ManualOpen := "DO_FaceplateDb".Cv38.ValveOpen;
	"MV3000LineAnimationDb"."Node 28".V08.ManualOpen := "DO_FaceplateDb".Cv46.ValveOpen;
	"MV3000LineAnimationDb"."Node 28".V09.ManualOpen := "DO_FaceplateDb".Cv52.ValveOpen;
	"MV3000LineAnimationDb"."Node 28".V10.ManualOpen := "DO_FaceplateDb".Cv58.ValveOpen;
	"MV3000LineAnimationDb"."Node 28".V11.ManualOpen := "DO_FaceplateDb".Cv59.ValveOpen;
	
	"MV3000LineAnimationDb"."Node 29".V01.ManualOpen := "DO_FaceplateDb".Cv04.ValveOpen;
	"MV3000LineAnimationDb"."Node 29".V02.ManualOpen := "DO_FaceplateDb".Cv01.ValveOpen;
	
	"MV3000LineAnimationDb"."Node 30".V01.ManualOpen := "DO_FaceplateDb".Cv06.ValveOpen;
	"MV3000LineAnimationDb"."Node 30".V02.ManualOpen := "DO_FaceplateDb".Cv09.ValveOpen;
	
	"MV3000LineAnimationDb"."Node31".V01.ManualOpen := "DO_FaceplateDb".Cv06.ValveOpen;
	"MV3000LineAnimationDb"."Node31".V02.ManualOpen := "DO_FaceplateDb".Cv09.ValveOpen;
	"MV3000LineAnimationDb"."Node31".V03.ManualOpen := "DO_FaceplateDb".Cv08.ValveOpen;
	
	
	"MV3000LineAnimationDb".Node32.V01.ManualOpen := "DO_FaceplateDb".Cv05.ValveOpen;
	"MV3000LineAnimationDb".Node32.V02.ManualOpen := "DO_FaceplateDb".Cv24.ValveOpen;
	
	"MV3000LineAnimationDb".Node33.V01.ManualOpen := "DO_FaceplateDb".Fbov01.ValveOpen;
	"MV3000LineAnimationDb".Node33.V02.ManualOpen := "DO_FaceplateDb".Cv26.ValveOpen;
	
	"MV3000LineAnimationDb".Node34.V01.ManualOpen := "DO_FaceplateDb".Cv42.ValveOpen;
	"MV3000LineAnimationDb".Node34.V02.ManualOpen := "DO_FaceplateDb".Cv54.ValveOpen;
	"MV3000LineAnimationDb".Node34.V03.ManualOpen := "DO_FaceplateDb".Cv48.ValveOpen;
	
	
	
END_FUNCTION

FUNCTION "BatchSA" : Void   // FC301, LAD
{ S7_Optimized_Access := 'TRUE' }
// stored: AutoNumber false, SetENOAutomatically false
   VAR_TEMP   // added for the SCL form of the ladder/FBD networks
      _w1 : Bool;
      _w2 : Bool;
      _w3 : Bool;
   END_VAR
BEGIN

REGION Network 1: "BatchSAD".Fault
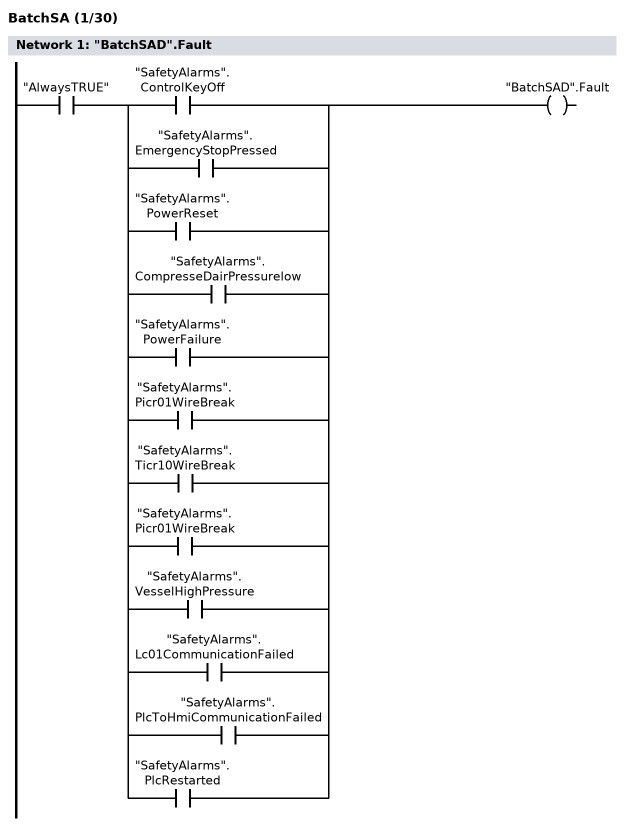
   RUNG wire#powerrail
      Contact( "AlwaysTRUE" )
      wire#w1
      Contact( "SafetyAlarms".ControlKeyOff )
      wire#w2
      Coil( "BatchSAD".Fault )
   END_RUNG
   RUNG wire#w1
      Contact( "SafetyAlarms".EmergencyStopPressed )
   END_RUNG wire#w2
   RUNG wire#w1
      Contact( "SafetyAlarms".PowerReset )
   END_RUNG wire#w2
   RUNG wire#w1
      Contact( "SafetyAlarms".CompresseDairPressurelow )
   END_RUNG wire#w2
   RUNG wire#w1
      Contact( "SafetyAlarms".PowerFailure )
   END_RUNG wire#w2
   RUNG wire#w1
      Contact( "SafetyAlarms".Picr01WireBreak )
   END_RUNG wire#w2
   RUNG wire#w1
      Contact( "SafetyAlarms".Ticr10WireBreak )
   END_RUNG wire#w2
   RUNG wire#w1
      Contact( "SafetyAlarms".Picr01WireBreak )
   END_RUNG wire#w2
   RUNG wire#w1
      Contact( "SafetyAlarms".VesselHighPressure )
   END_RUNG wire#w2
   RUNG wire#w1
      Contact( "SafetyAlarms".Lc01CommunicationFailed )
   END_RUNG wire#w2
   RUNG wire#w1
      Contact( "SafetyAlarms".PlcToHmiCommunicationFailed )
   END_RUNG wire#w2
   RUNG wire#w1
      Contact( "SafetyAlarms".PlcRestarted )
   END_RUNG wire#w2
   // the same network as SCL:
   "BatchSAD".Fault := "AlwaysTRUE" AND ("SafetyAlarms".ControlKeyOff OR "SafetyAlarms".EmergencyStopPressed OR "SafetyAlarms".PowerReset OR "SafetyAlarms".CompresseDairPressurelow OR "SafetyAlarms".PowerFailure OR "SafetyAlarms".Picr01WireBreak OR "SafetyAlarms".Ticr10WireBreak OR "SafetyAlarms".Picr01WireBreak OR "SafetyAlarms".VesselHighPressure OR "SafetyAlarms".Lc01CommunicationFailed OR "SafetyAlarms".PlcToHmiCommunicationFailed OR "SafetyAlarms".PlcRestarted);
END_REGION

REGION Network 2: Batch Selected
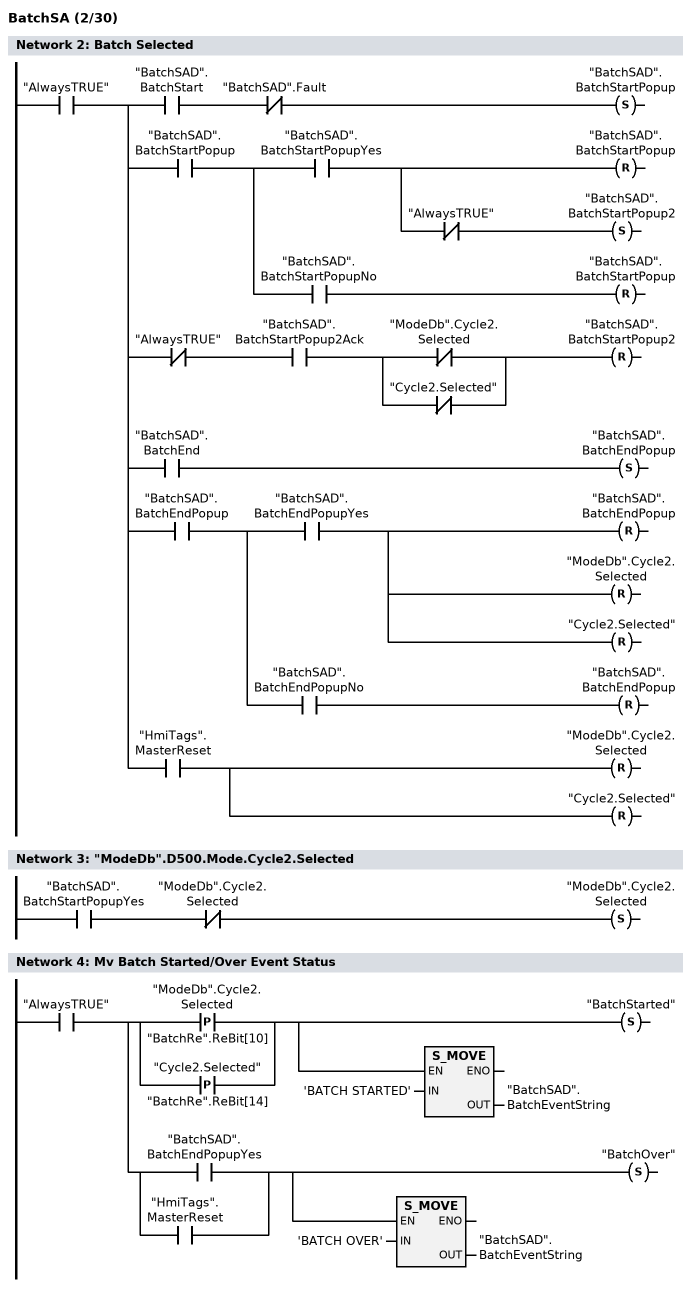
   RUNG wire#powerrail
      Contact( "AlwaysTRUE" )
      wire#w1
      Contact( "BatchSAD".BatchStart )
      I_Contact( "BatchSAD".Fault )
      S_Coil( "BatchSAD".BatchStartPopup )
   END_RUNG
   RUNG wire#w1
      Contact( "BatchSAD".BatchStartPopup )
      wire#w2
      Contact( "BatchSAD".BatchStartPopupYes )
      wire#w3
      R_Coil( "BatchSAD".BatchStartPopup )
   END_RUNG
   RUNG wire#w3
      I_Contact( "AlwaysTRUE" )
      S_Coil( "BatchSAD".BatchStartPopup2 )
   END_RUNG
   RUNG wire#w2
      Contact( "BatchSAD".BatchStartPopupNo )
      R_Coil( "BatchSAD".BatchStartPopup )
   END_RUNG
   RUNG wire#w1
      I_Contact( "AlwaysTRUE" )
      Contact( "BatchSAD".BatchStartPopup2Ack )
      wire#w4
      I_Contact( "ModeDb".Cycle2.Selected )
      wire#w5
      R_Coil( "BatchSAD".BatchStartPopup2 )
   END_RUNG
   RUNG wire#w4
      I_Contact( "Cycle2.Selected" )
   END_RUNG wire#w5
   RUNG wire#w1
      Contact( "BatchSAD".BatchEnd )
      S_Coil( "BatchSAD".BatchEndPopup )
   END_RUNG
   RUNG wire#w1
      Contact( "BatchSAD".BatchEndPopup )
      wire#w6
      Contact( "BatchSAD".BatchEndPopupYes )
      wire#w7
      R_Coil( "BatchSAD".BatchEndPopup )
   END_RUNG
   RUNG wire#w7
      R_Coil( "ModeDb".Cycle2.Selected )
   END_RUNG
   RUNG wire#w7
      R_Coil( "Cycle2.Selected" )
   END_RUNG
   RUNG wire#w6
      Contact( "BatchSAD".BatchEndPopupNo )
      R_Coil( "BatchSAD".BatchEndPopup )
   END_RUNG
   RUNG wire#w1
      Contact( "HmiTags".MasterReset )
      wire#w8
      R_Coil( "ModeDb".Cycle2.Selected )
   END_RUNG
   RUNG wire#w8
      R_Coil( "Cycle2.Selected" )
   END_RUNG
   // the same network as SCL:
   IF "AlwaysTRUE" AND "BatchSAD".BatchStart AND NOT "BatchSAD".Fault THEN
       "BatchSAD".BatchStartPopup := TRUE;
   END_IF;
   #_w1 := "AlwaysTRUE" AND "BatchSAD".BatchStartPopup;
   #_w2 := #_w1 AND "BatchSAD".BatchStartPopupYes;
   IF #_w2 THEN "BatchSAD".BatchStartPopup := FALSE; END_IF;
   IF #_w2 AND NOT "AlwaysTRUE" THEN "BatchSAD".BatchStartPopup2 := TRUE; END_IF;
   IF #_w1 AND "BatchSAD".BatchStartPopupNo THEN "BatchSAD".BatchStartPopup := FALSE; END_IF;
   IF "AlwaysTRUE" AND NOT "AlwaysTRUE" AND "BatchSAD".BatchStartPopup2Ack AND (NOT "ModeDb".Cycle2.Selected OR NOT "Cycle2.Selected") THEN
       "BatchSAD".BatchStartPopup2 := FALSE;
   END_IF;
   IF "AlwaysTRUE" AND "BatchSAD".BatchEnd THEN "BatchSAD".BatchEndPopup := TRUE; END_IF;
   #_w3 := "AlwaysTRUE" AND "BatchSAD".BatchEndPopup;
   IF #_w3 AND "BatchSAD".BatchEndPopupYes THEN
       "BatchSAD".BatchEndPopup := FALSE;
       "ModeDb".Cycle2.Selected := FALSE;
       "Cycle2.Selected" := FALSE;
   END_IF;
   IF #_w3 AND "BatchSAD".BatchEndPopupNo THEN "BatchSAD".BatchEndPopup := FALSE; END_IF;
   IF "AlwaysTRUE" AND "HmiTags".MasterReset THEN
       "ModeDb".Cycle2.Selected := FALSE;
       "Cycle2.Selected" := FALSE;
   END_IF;
END_REGION

REGION Network 3: "ModeDb".D500.Mode.Cycle2.Selected
   RUNG wire#powerrail
      Contact( "BatchSAD".BatchStartPopupYes )
      I_Contact( "ModeDb".Cycle2.Selected )
      S_Coil( "ModeDb".Cycle2.Selected )
   END_RUNG
   // the same network as SCL:
   IF "BatchSAD".BatchStartPopupYes AND NOT "ModeDb".Cycle2.Selected THEN
       "ModeDb".Cycle2.Selected := TRUE;
   END_IF;
END_REGION

REGION Network 4: Mv Batch Started/Over Event Status
   RUNG wire#powerrail
      Contact( "AlwaysTRUE" )
      wire#w1
      P_Contact(operand := "ModeDb".Cycle2.Selected, bit := "BatchRe".ReBit[10])
      wire#w2
      S_Coil( "BatchStarted" )
   END_RUNG
   RUNG wire#w1
      P_Contact(operand := "Cycle2.Selected", bit := "BatchRe".ReBit[14])
   END_RUNG wire#w2
   RUNG wire#w2
      S_Move(in := 'BATCH STARTED', out => "BatchSAD".BatchEventString)
   END_RUNG
   RUNG wire#w1
      Contact( "BatchSAD".BatchEndPopupYes )
      wire#w3
      S_Coil( "BatchOver" )
   END_RUNG
   RUNG wire#w1
      Contact( "HmiTags".MasterReset )
   END_RUNG wire#w3
   RUNG wire#w3
      S_Move(in := 'BATCH OVER', out => "BatchSAD".BatchEventString)
   END_RUNG
   // the same network as SCL:
   #_w1 := "AlwaysTRUE" AND "ModeDb".Cycle2.Selected AND NOT "BatchRe".ReBit[10];   // rising edge of "ModeDb".Cycle2.Selected
   "BatchRe".ReBit[10] := "ModeDb".Cycle2.Selected;
   #_w2 := "AlwaysTRUE" AND "Cycle2.Selected" AND NOT "BatchRe".ReBit[14];   // rising edge of "Cycle2.Selected"
   "BatchRe".ReBit[14] := "Cycle2.Selected";
   IF #_w1 OR #_w2 THEN
       "BatchStarted" := TRUE;
       "BatchSAD".BatchEventString := 'BATCH STARTED';
   END_IF;
   IF "AlwaysTRUE" AND ("BatchSAD".BatchEndPopupYes OR "HmiTags".MasterReset) THEN
       "BatchOver" := TRUE;
       "BatchSAD".BatchEventString := 'BATCH OVER';
   END_IF;
END_REGION

REGION Network 5: Mv Batch Started/Over Event Status
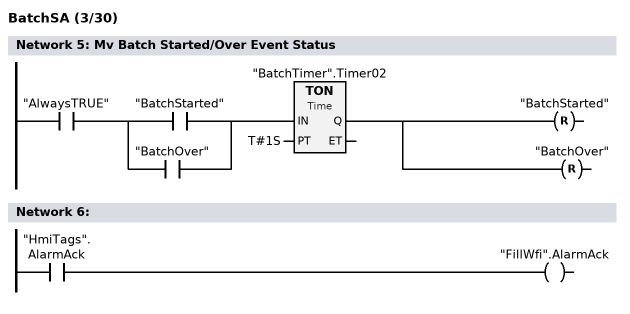
   RUNG wire#powerrail
      Contact( "AlwaysTRUE" )
      wire#w1
      Contact( "BatchStarted" )
      wire#w2
      { S7_Templates := "time_type := Time" } "BatchTimer".Timer02.TON(pt := T#1S, et =>)
      wire#w3
      R_Coil( "BatchStarted" )
   END_RUNG
   RUNG wire#w1
      Contact( "BatchOver" )
   END_RUNG wire#w2
   RUNG wire#w3
      R_Coil( "BatchOver" )
   END_RUNG
   // the same network as SCL:
   "BatchTimer".Timer02.TON(IN := "AlwaysTRUE" AND ("BatchStarted" OR "BatchOver"), PT := T#1S);
   IF "BatchTimer".Timer02.Q THEN
       "BatchStarted" := FALSE;
       "BatchOver" := FALSE;
   END_IF;
END_REGION

REGION Network 6
   RUNG wire#powerrail
      Contact( "HmiTags".AlarmAck )
      Coil( "FillWfi".AlarmAck )
   END_RUNG
   // the same network as SCL:
   "FillWfi".AlarmAck := "HmiTags".AlarmAck;
END_REGION

REGION Network 7: ******************************Fill Wfi******************************
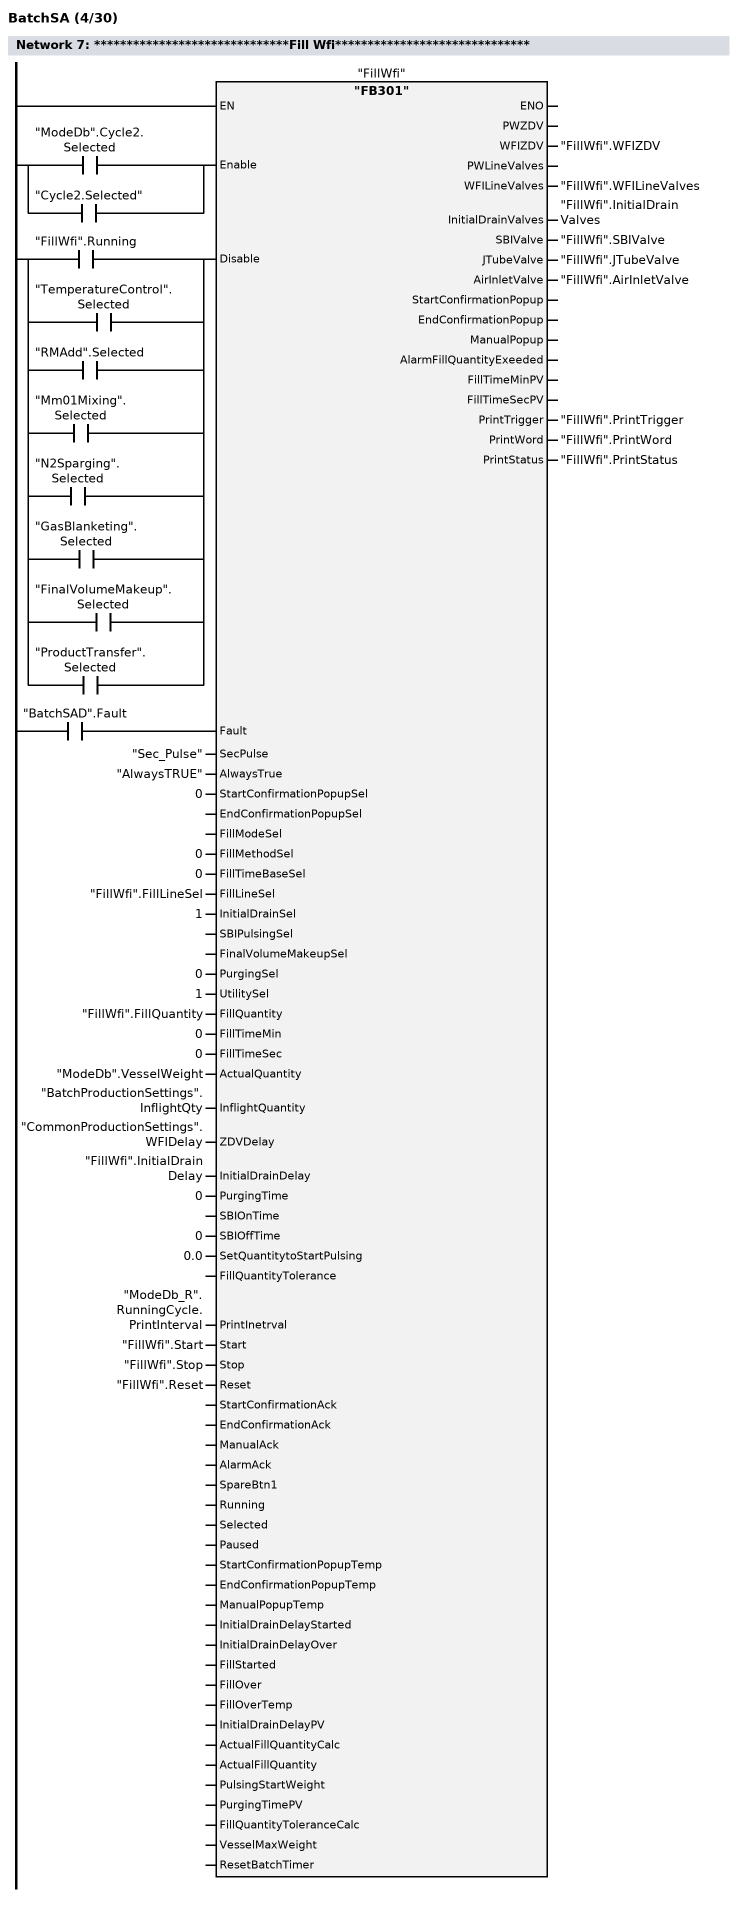
   RUNG wire#powerrail
      "FillWfi"(Enable := wire#w1, Disable := wire#w2, Fault := wire#w3, SecPulse := "Sec_Pulse", AlwaysTrue := "AlwaysTRUE", StartConfirmationPopupSel := 0, EndConfirmationPopupSel :=, FillModeSel :=, FillMethodSel := 0, FillTimeBaseSel := 0, FillLineSel := "FillWfi".FillLineSel, InitialDrainSel := 1, SBIPulsingSel :=, FinalVolumeMakeupSel :=, PurgingSel := 0, UtilitySel := 1, FillQuantity := "FillWfi".FillQuantity, FillTimeMin := 0, FillTimeSec := 0, ActualQuantity := "ModeDb".VesselWeight, InflightQuantity := "BatchProductionSettings".InflightQty, ZDVDelay := "CommonProductionSettings".WFIDelay, InitialDrainDelay := "FillWfi".InitialDrainDelay, PurgingTime := 0, SBIOnTime :=, SBIOffTime := 0, SetQuantitytoStartPulsing := 0.0, FillQuantityTolerance :=, PrintInetrval := "ModeDb_R".RunningCycle.PrintInterval, Start := "FillWfi".Start, Stop := "FillWfi".Stop, Reset := "FillWfi".Reset, StartConfirmationAck :=, EndConfirmationAck :=, ManualAck :=, AlarmAck :=, SpareBtn1 :=, Running :=, Selected :=, Paused :=, StartConfirmationPopupTemp :=, EndConfirmationPopupTemp :=, ManualPopupTemp :=, InitialDrainDelayStarted :=, InitialDrainDelayOver :=, FillStarted :=, FillOver :=, FillOverTemp :=, InitialDrainDelayPV :=, ActualFillQuantityCalc :=, ActualFillQuantity :=, PulsingStartWeight :=, PurgingTimePV :=, FillQuantityToleranceCalc :=, VesselMaxWeight :=, ResetBatchTimer :=, PWZDV =>, WFIZDV => "FillWfi".WFIZDV, PWLineValves =>, WFILineValves => "FillWfi".WFILineValves, InitialDrainValves => "FillWfi".InitialDrainValves, SBIValve => "FillWfi".SBIValve, JTubeValve => "FillWfi".JTubeValve, AirInletValve => "FillWfi".AirInletValve, StartConfirmationPopup =>, EndConfirmationPopup =>, ManualPopup =>, AlarmFillQuantityExeeded =>, FillTimeMinPV =>, FillTimeSecPV =>, PrintTrigger => "FillWfi".PrintTrigger, PrintWord => "FillWfi".PrintWord, PrintStatus => "FillWfi".PrintStatus)
   END_RUNG
   RUNG wire#powerrail
      Contact( "ModeDb".Cycle2.Selected )
   END_RUNG wire#w1
   RUNG wire#powerrail
      Contact( "Cycle2.Selected" )
   END_RUNG wire#w1
   RUNG wire#powerrail
      Contact( "FillWfi".Running )
   END_RUNG wire#w2
   RUNG wire#powerrail
      Contact( "TemperatureControl".Selected )
   END_RUNG wire#w2
   RUNG wire#powerrail
      Contact( "RMAdd".Selected )
   END_RUNG wire#w2
   RUNG wire#powerrail
      Contact( "Mm01Mixing".Selected )
   END_RUNG wire#w2
   RUNG wire#powerrail
      Contact( "N2Sparging".Selected )
   END_RUNG wire#w2
   RUNG wire#powerrail
      Contact( "GasBlanketing".Selected )
   END_RUNG wire#w2
   RUNG wire#powerrail
      Contact( "FinalVolumeMakeup".Selected )
   END_RUNG wire#w2
   RUNG wire#powerrail
      Contact( "ProductTransfer".Selected )
   END_RUNG wire#w2
   RUNG wire#powerrail
      Contact( "BatchSAD".Fault )
   END_RUNG wire#w3
   // the same network as SCL:
   "FillWfi"(Enable := "ModeDb".Cycle2.Selected OR "Cycle2.Selected",   // "FB301"
             Disable := "FillWfi".Running OR "TemperatureControl".Selected OR "RMAdd".Selected OR "Mm01Mixing".Selected OR "N2Sparging".Selected OR "GasBlanketing".Selected OR "FinalVolumeMakeup".Selected OR "ProductTransfer".Selected,
             Fault := "BatchSAD".Fault,
             SecPulse := "Sec_Pulse",
             AlwaysTrue := "AlwaysTRUE",
             StartConfirmationPopupSel := 0,
             FillMethodSel := 0,
             FillTimeBaseSel := 0,
             FillLineSel := "FillWfi".FillLineSel,
             InitialDrainSel := 1,
             PurgingSel := 0,
             UtilitySel := 1,
             FillQuantity := "FillWfi".FillQuantity,
             FillTimeMin := 0,
             FillTimeSec := 0,
             ActualQuantity := "ModeDb".VesselWeight,
             InflightQuantity := "BatchProductionSettings".InflightQty,
             ZDVDelay := "CommonProductionSettings".WFIDelay,
             InitialDrainDelay := "FillWfi".InitialDrainDelay,
             PurgingTime := 0,
             SBIOffTime := 0,
             SetQuantitytoStartPulsing := 0.0,
             PrintInetrval := "ModeDb_R".RunningCycle.PrintInterval,
             Start := "FillWfi".Start,
             Stop := "FillWfi".Stop,
             Reset := "FillWfi".Reset,
             WFIZDV => "FillWfi".WFIZDV,
             WFILineValves => "FillWfi".WFILineValves,
             InitialDrainValves => "FillWfi".InitialDrainValves,
             SBIValve => "FillWfi".SBIValve,
             JTubeValve => "FillWfi".JTubeValve,
             AirInletValve => "FillWfi".AirInletValve,
             PrintTrigger => "FillWfi".PrintTrigger,
             PrintWord => "FillWfi".PrintWord,
             PrintStatus => "FillWfi".PrintStatus);
END_REGION

REGION Network 8: Fill Wfi Events
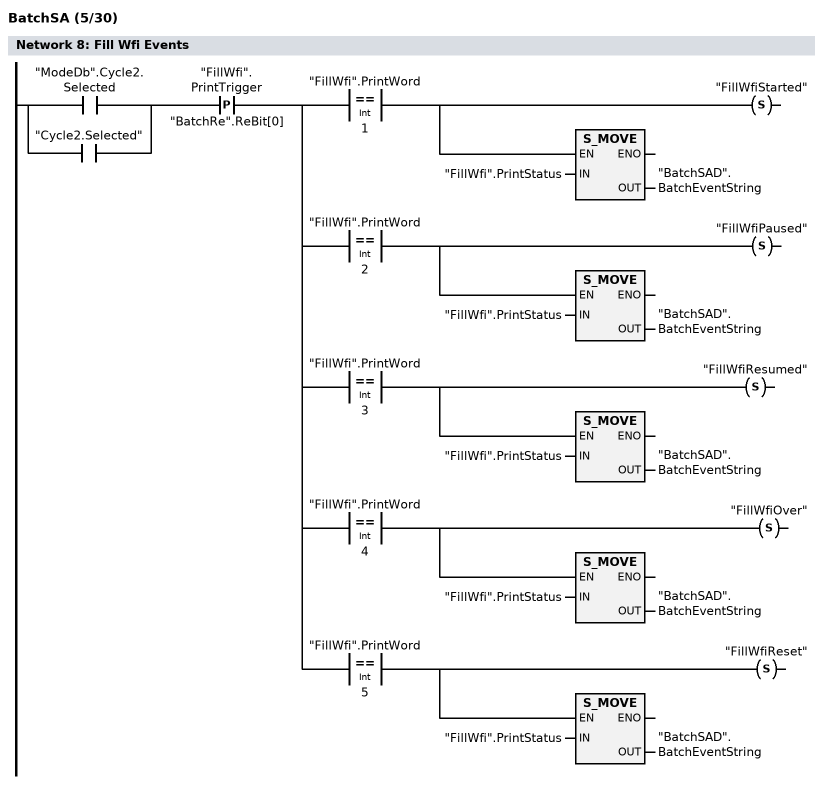
   RUNG wire#powerrail
      Contact( "ModeDb".Cycle2.Selected )
      wire#w1
      P_Contact(operand := "FillWfi".PrintTrigger, bit := "BatchRe".ReBit[0])
      wire#w2
      { S7_Templates := "SrcType := Int" } EQ_Contact(in1 := "FillWfi".PrintWord, in2 := 1)
      wire#w3
      S_Coil( "FillWfiStarted" )
   END_RUNG
   RUNG wire#powerrail
      Contact( "Cycle2.Selected" )
   END_RUNG wire#w1
   RUNG wire#w3
      S_Move(in := "FillWfi".PrintStatus, out => "BatchSAD".BatchEventString)
   END_RUNG
   RUNG wire#w2
      { S7_Templates := "SrcType := Int" } EQ_Contact(in1 := "FillWfi".PrintWord, in2 := 2)
      wire#w4
      S_Coil( "FillWfiPaused" )
   END_RUNG
   RUNG wire#w4
      S_Move(in := "FillWfi".PrintStatus, out => "BatchSAD".BatchEventString)
   END_RUNG
   RUNG wire#w2
      { S7_Templates := "SrcType := Int" } EQ_Contact(in1 := "FillWfi".PrintWord, in2 := 3)
      wire#w5
      S_Coil( "FillWfiResumed" )
   END_RUNG
   RUNG wire#w5
      S_Move(in := "FillWfi".PrintStatus, out => "BatchSAD".BatchEventString)
   END_RUNG
   RUNG wire#w2
      { S7_Templates := "SrcType := Int" } EQ_Contact(in1 := "FillWfi".PrintWord, in2 := 4)
      wire#w6
      S_Coil( "FillWfiOver" )
   END_RUNG
   RUNG wire#w6
      S_Move(in := "FillWfi".PrintStatus, out => "BatchSAD".BatchEventString)
   END_RUNG
   RUNG wire#w2
      { S7_Templates := "SrcType := Int" } EQ_Contact(in1 := "FillWfi".PrintWord, in2 := 5)
      wire#w7
      S_Coil( "FillWfiReset" )
   END_RUNG
   RUNG wire#w7
      S_Move(in := "FillWfi".PrintStatus, out => "BatchSAD".BatchEventString)
   END_RUNG
   // the same network as SCL:
   #_w1 := ("ModeDb".Cycle2.Selected OR "Cycle2.Selected") AND "FillWfi".PrintTrigger AND NOT "BatchRe".ReBit[0];   // rising edge of "FillWfi".PrintTrigger
   "BatchRe".ReBit[0] := "FillWfi".PrintTrigger;
   IF #_w1 AND ("FillWfi".PrintWord = 1) THEN
       "FillWfiStarted" := TRUE;
       "BatchSAD".BatchEventString := "FillWfi".PrintStatus;
   END_IF;
   IF #_w1 AND ("FillWfi".PrintWord = 2) THEN
       "FillWfiPaused" := TRUE;
       "BatchSAD".BatchEventString := "FillWfi".PrintStatus;
   END_IF;
   IF #_w1 AND ("FillWfi".PrintWord = 3) THEN
       "FillWfiResumed" := TRUE;
       "BatchSAD".BatchEventString := "FillWfi".PrintStatus;
   END_IF;
   IF #_w1 AND ("FillWfi".PrintWord = 4) THEN
       "FillWfiOver" := TRUE;
       "BatchSAD".BatchEventString := "FillWfi".PrintStatus;
   END_IF;
   IF #_w1 AND ("FillWfi".PrintWord = 5) THEN
       "FillWfiReset" := TRUE;
       "BatchSAD".BatchEventString := "FillWfi".PrintStatus;
   END_IF;
END_REGION

REGION Network 9: ******************************Temperature Control******************************
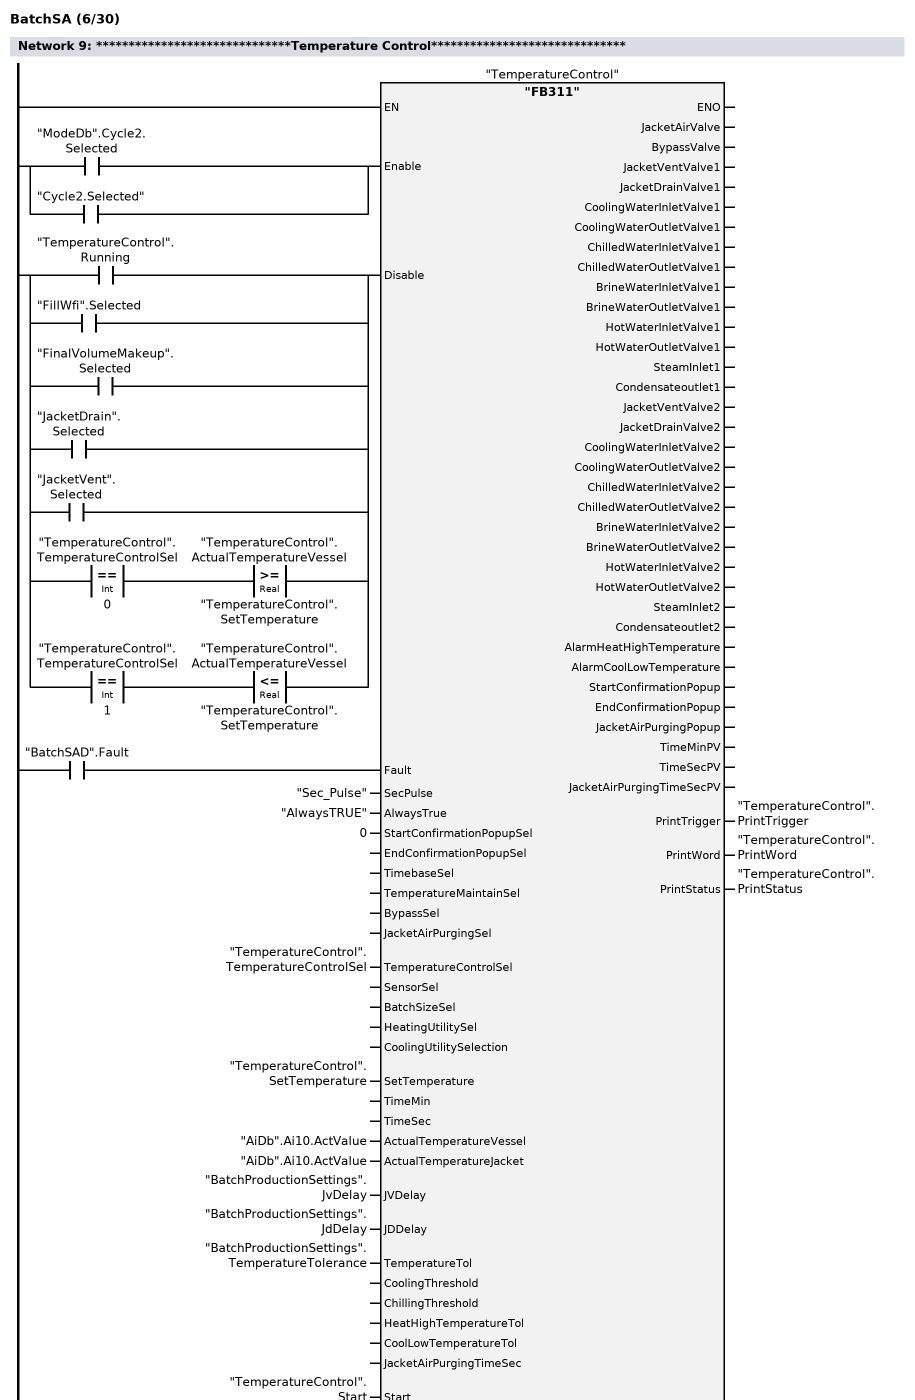
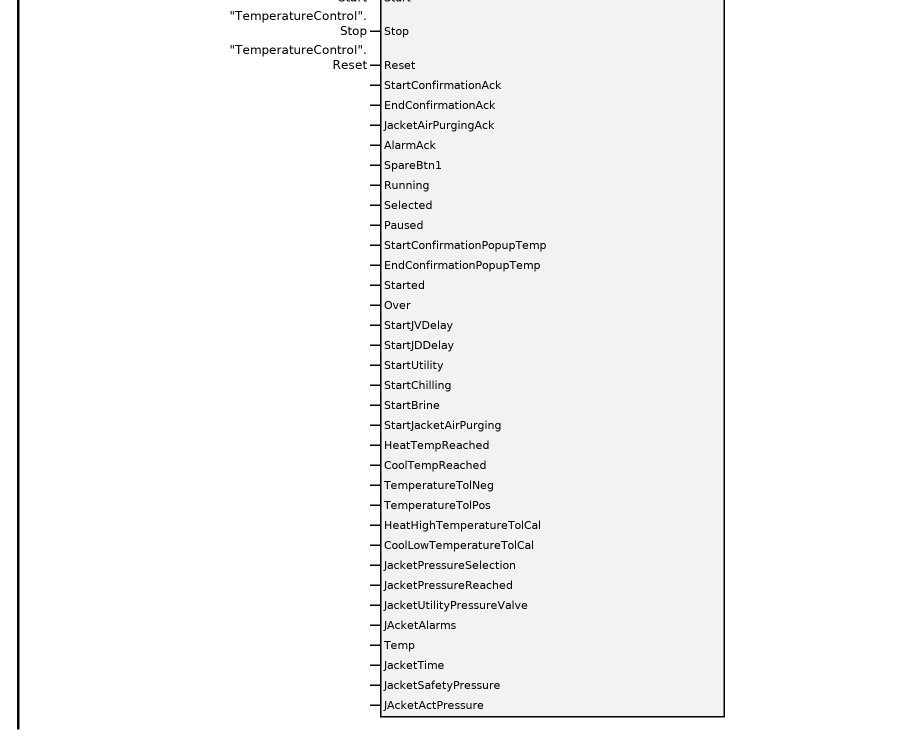
   RUNG wire#powerrail
      "TemperatureControl"(Enable := wire#w1, Disable := wire#w2, Fault := wire#w3, SecPulse := "Sec_Pulse", AlwaysTrue := "AlwaysTRUE", StartConfirmationPopupSel := 0, EndConfirmationPopupSel :=, TimebaseSel :=, TemperatureMaintainSel :=, BypassSel :=, JacketAirPurgingSel :=, TemperatureControlSel := "TemperatureControl".TemperatureControlSel, SensorSel :=, BatchSizeSel :=, HeatingUtilitySel :=, CoolingUtilitySelection :=, SetTemperature := "TemperatureControl".SetTemperature, TimeMin :=, TimeSec :=, ActualTemperatureVessel := "AiDb".Ai10.ActValue, ActualTemperatureJacket := "AiDb".Ai10.ActValue, JVDelay := "BatchProductionSettings".JvDelay, JDDelay := "BatchProductionSettings".JdDelay, TemperatureTol := "BatchProductionSettings".TemperatureTolerance, CoolingThreshold :=, ChillingThreshold :=, HeatHighTemperatureTol :=, CoolLowTemperatureTol :=, JacketAirPurgingTimeSec :=, Start := "TemperatureControl".Start, Stop := "TemperatureControl".Stop, Reset := "TemperatureControl".Reset, StartConfirmationAck :=, EndConfirmationAck :=, JacketAirPurgingAck :=, AlarmAck :=, SpareBtn1 :=, Running :=, Selected :=, Paused :=, StartConfirmationPopupTemp :=, EndConfirmationPopupTemp :=, Started :=, Over :=, StartJVDelay :=, StartJDDelay :=, StartUtility :=, StartChilling :=, StartBrine :=, StartJacketAirPurging :=, HeatTempReached :=, CoolTempReached :=, TemperatureTolNeg :=, TemperatureTolPos :=, HeatHighTemperatureTolCal :=, CoolLowTemperatureTolCal :=, JacketPressureSelection :=, JacketPressureReached :=, JacketUtilityPressureValve :=, JAcketAlarms :=, Temp :=, JacketTime :=, JacketSafetyPressure :=, JAcketActPressure :=, JacketAirValve =>, BypassValve =>, JacketVentValve1 =>, JacketDrainValve1 =>, CoolingWaterInletValve1 =>, CoolingWaterOutletValve1 =>, ChilledWaterInletValve1 =>, ChilledWaterOutletValve1 =>, BrineWaterInletValve1 =>, BrineWaterOutletValve1 =>, HotWaterInletValve1 =>, HotWaterOutletValve1 =>, SteamInlet1 =>, Condensateoutlet1 =>, JacketVentValve2 =>, JacketDrainValve2 =>, CoolingWaterInletValve2 =>, CoolingWaterOutletValve2 =>, ChilledWaterInletValve2 =>, ChilledWaterOutletValve2 =>, BrineWaterInletValve2 =>, BrineWaterOutletValve2 =>, HotWaterInletValve2 =>, HotWaterOutletValve2 =>, SteamInlet2 =>, Condensateoutlet2 =>, AlarmHeatHighTemperature =>, AlarmCoolLowTemperature =>, StartConfirmationPopup =>, EndConfirmationPopup =>, JacketAirPurgingPopup =>, TimeMinPV =>, TimeSecPV =>, JacketAirPurgingTimeSecPV =>, PrintTrigger => "TemperatureControl".PrintTrigger, PrintWord => "TemperatureControl".PrintWord, PrintStatus => "TemperatureControl".PrintStatus)
   END_RUNG
   RUNG wire#powerrail
      Contact( "ModeDb".Cycle2.Selected )
   END_RUNG wire#w1
   RUNG wire#powerrail
      Contact( "Cycle2.Selected" )
   END_RUNG wire#w1
   RUNG wire#powerrail
      Contact( "TemperatureControl".Running )
   END_RUNG wire#w2
   RUNG wire#powerrail
      Contact( "FillWfi".Selected )
   END_RUNG wire#w2
   RUNG wire#powerrail
      Contact( "FinalVolumeMakeup".Selected )
   END_RUNG wire#w2
   RUNG wire#powerrail
      Contact( "JacketDrain".Selected )
   END_RUNG wire#w2
   RUNG wire#powerrail
      Contact( "JacketVent".Selected )
   END_RUNG wire#w2
   RUNG wire#powerrail
      { S7_Templates := "SrcType := Int" } EQ_Contact(in1 := "TemperatureControl".TemperatureControlSel, in2 := 0)
      { S7_Templates := "SrcType := Real" } GE_Contact(in1 := "TemperatureControl".ActualTemperatureVessel, in2 := "TemperatureControl".SetTemperature)
   END_RUNG wire#w2
   RUNG wire#powerrail
      { S7_Templates := "SrcType := Int" } EQ_Contact(in1 := "TemperatureControl".TemperatureControlSel, in2 := 1)
      { S7_Templates := "SrcType := Real" } LE_Contact(in1 := "TemperatureControl".ActualTemperatureVessel, in2 := "TemperatureControl".SetTemperature)
   END_RUNG wire#w2
   RUNG wire#powerrail
      Contact( "BatchSAD".Fault )
   END_RUNG wire#w3
   // the same network as SCL:
   "TemperatureControl"(Enable := "ModeDb".Cycle2.Selected OR "Cycle2.Selected",   // "FB311"
                        Disable := "TemperatureControl".Running OR "FillWfi".Selected OR "FinalVolumeMakeup".Selected OR "JacketDrain".Selected OR "JacketVent".Selected OR (("TemperatureControl".TemperatureControlSel = 0) AND ("TemperatureControl".ActualTemperatureVessel >= "TemperatureControl".SetTemperature)) OR (("TemperatureControl".TemperatureControlSel = 1) AND ("TemperatureControl".ActualTemperatureVessel <= "TemperatureControl".SetTemperature)),
                        Fault := "BatchSAD".Fault,
                        SecPulse := "Sec_Pulse",
                        AlwaysTrue := "AlwaysTRUE",
                        StartConfirmationPopupSel := 0,
                        TemperatureControlSel := "TemperatureControl".TemperatureControlSel,
                        SetTemperature := "TemperatureControl".SetTemperature,
                        ActualTemperatureVessel := "AiDb".Ai10.ActValue,
                        ActualTemperatureJacket := "AiDb".Ai10.ActValue,
                        JVDelay := "BatchProductionSettings".JvDelay,
                        JDDelay := "BatchProductionSettings".JdDelay,
                        TemperatureTol := "BatchProductionSettings".TemperatureTolerance,
                        Start := "TemperatureControl".Start,
                        Stop := "TemperatureControl".Stop,
                        Reset := "TemperatureControl".Reset,
                        PrintTrigger => "TemperatureControl".PrintTrigger,
                        PrintWord => "TemperatureControl".PrintWord,
                        PrintStatus => "TemperatureControl".PrintStatus);
END_REGION

REGION Network 10: Temprature Control Event Status
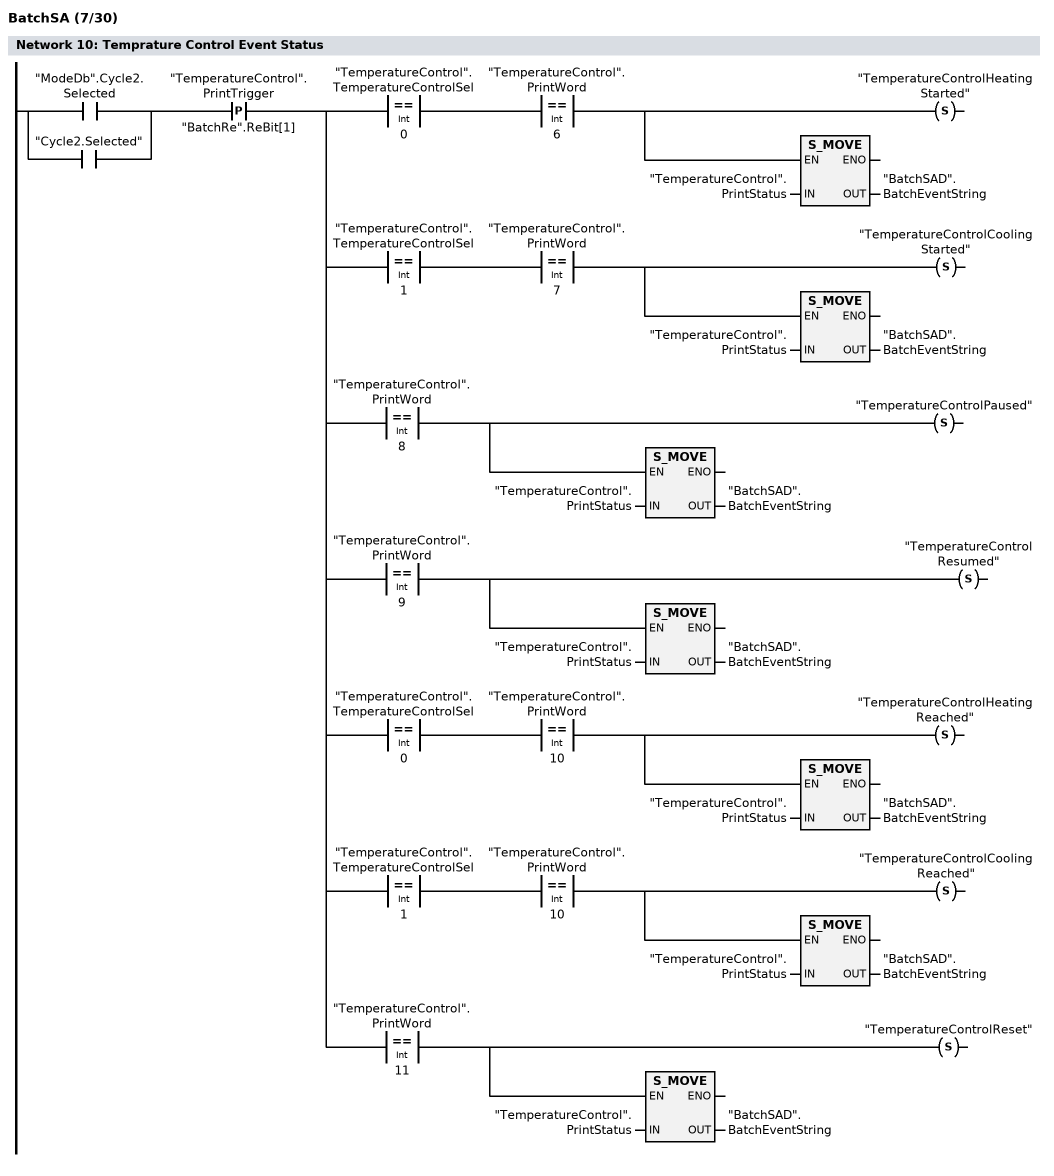
   RUNG wire#powerrail
      Contact( "ModeDb".Cycle2.Selected )
      wire#w1
      P_Contact(operand := "TemperatureControl".PrintTrigger, bit := "BatchRe".ReBit[1])
      wire#w2
      { S7_Templates := "SrcType := Int" } EQ_Contact(in1 := "TemperatureControl".TemperatureControlSel, in2 := 0)
      { S7_Templates := "SrcType := Int" } EQ_Contact(in1 := "TemperatureControl".PrintWord, in2 := 6)
      wire#w3
      S_Coil( "TemperatureControlHeatingStarted" )
   END_RUNG
   RUNG wire#powerrail
      Contact( "Cycle2.Selected" )
   END_RUNG wire#w1
   RUNG wire#w3
      S_Move(in := "TemperatureControl".PrintStatus, out => "BatchSAD".BatchEventString)
   END_RUNG
   RUNG wire#w2
      { S7_Templates := "SrcType := Int" } EQ_Contact(in1 := "TemperatureControl".TemperatureControlSel, in2 := 1)
      { S7_Templates := "SrcType := Int" } EQ_Contact(in1 := "TemperatureControl".PrintWord, in2 := 7)
      wire#w4
      S_Coil( "TemperatureControlCoolingStarted" )
   END_RUNG
   RUNG wire#w4
      S_Move(in := "TemperatureControl".PrintStatus, out => "BatchSAD".BatchEventString)
   END_RUNG
   RUNG wire#w2
      { S7_Templates := "SrcType := Int" } EQ_Contact(in1 := "TemperatureControl".PrintWord, in2 := 8)
      wire#w5
      S_Coil( "TemperatureControlPaused" )
   END_RUNG
   RUNG wire#w5
      S_Move(in := "TemperatureControl".PrintStatus, out => "BatchSAD".BatchEventString)
   END_RUNG
   RUNG wire#w2
      { S7_Templates := "SrcType := Int" } EQ_Contact(in1 := "TemperatureControl".PrintWord, in2 := 9)
      wire#w6
      S_Coil( "TemperatureControlResumed" )
   END_RUNG
   RUNG wire#w6
      S_Move(in := "TemperatureControl".PrintStatus, out => "BatchSAD".BatchEventString)
   END_RUNG
   RUNG wire#w2
      { S7_Templates := "SrcType := Int" } EQ_Contact(in1 := "TemperatureControl".TemperatureControlSel, in2 := 0)
      { S7_Templates := "SrcType := Int" } EQ_Contact(in1 := "TemperatureControl".PrintWord, in2 := 10)
      wire#w7
      S_Coil( "TemperatureControlHeatingReached" )
   END_RUNG
   RUNG wire#w7
      S_Move(in := "TemperatureControl".PrintStatus, out => "BatchSAD".BatchEventString)
   END_RUNG
   RUNG wire#w2
      { S7_Templates := "SrcType := Int" } EQ_Contact(in1 := "TemperatureControl".TemperatureControlSel, in2 := 1)
      { S7_Templates := "SrcType := Int" } EQ_Contact(in1 := "TemperatureControl".PrintWord, in2 := 10)
      wire#w8
      S_Coil( "TemperatureControlCoolingReached" )
   END_RUNG
   RUNG wire#w8
      S_Move(in := "TemperatureControl".PrintStatus, out => "BatchSAD".BatchEventString)
   END_RUNG
   RUNG wire#w2
      { S7_Templates := "SrcType := Int" } EQ_Contact(in1 := "TemperatureControl".PrintWord, in2 := 11)
      wire#w9
      S_Coil( "TemperatureControlReset" )
   END_RUNG
   RUNG wire#w9
      S_Move(in := "TemperatureControl".PrintStatus, out => "BatchSAD".BatchEventString)
   END_RUNG
   // the same network as SCL:
   #_w1 := ("ModeDb".Cycle2.Selected OR "Cycle2.Selected") AND "TemperatureControl".PrintTrigger AND NOT "BatchRe".ReBit[1];   // rising edge of "TemperatureControl".PrintTrigger
   "BatchRe".ReBit[1] := "TemperatureControl".PrintTrigger;
   IF #_w1 AND ("TemperatureControl".TemperatureControlSel = 0) AND ("TemperatureControl".PrintWord = 6) THEN
       "TemperatureControlHeatingStarted" := TRUE;
       "BatchSAD".BatchEventString := "TemperatureControl".PrintStatus;
   END_IF;
   IF #_w1 AND ("TemperatureControl".TemperatureControlSel = 1) AND ("TemperatureControl".PrintWord = 7) THEN
       "TemperatureControlCoolingStarted" := TRUE;
       "BatchSAD".BatchEventString := "TemperatureControl".PrintStatus;
   END_IF;
   IF #_w1 AND ("TemperatureControl".PrintWord = 8) THEN
       "TemperatureControlPaused" := TRUE;
       "BatchSAD".BatchEventString := "TemperatureControl".PrintStatus;
   END_IF;
   IF #_w1 AND ("TemperatureControl".PrintWord = 9) THEN
       "TemperatureControlResumed" := TRUE;
       "BatchSAD".BatchEventString := "TemperatureControl".PrintStatus;
   END_IF;
   IF #_w1 AND ("TemperatureControl".TemperatureControlSel = 0) AND ("TemperatureControl".PrintWord = 10) THEN
       "TemperatureControlHeatingReached" := TRUE;
       "BatchSAD".BatchEventString := "TemperatureControl".PrintStatus;
   END_IF;
   IF #_w1 AND ("TemperatureControl".TemperatureControlSel = 1) AND ("TemperatureControl".PrintWord = 10) THEN
       "TemperatureControlCoolingReached" := TRUE;
       "BatchSAD".BatchEventString := "TemperatureControl".PrintStatus;
   END_IF;
   IF #_w1 AND ("TemperatureControl".PrintWord = 11) THEN
       "TemperatureControlReset" := TRUE;
       "BatchSAD".BatchEventString := "TemperatureControl".PrintStatus;
   END_IF;
END_REGION

REGION Network 11: "BATCH TempControlBlock" - ON OFF
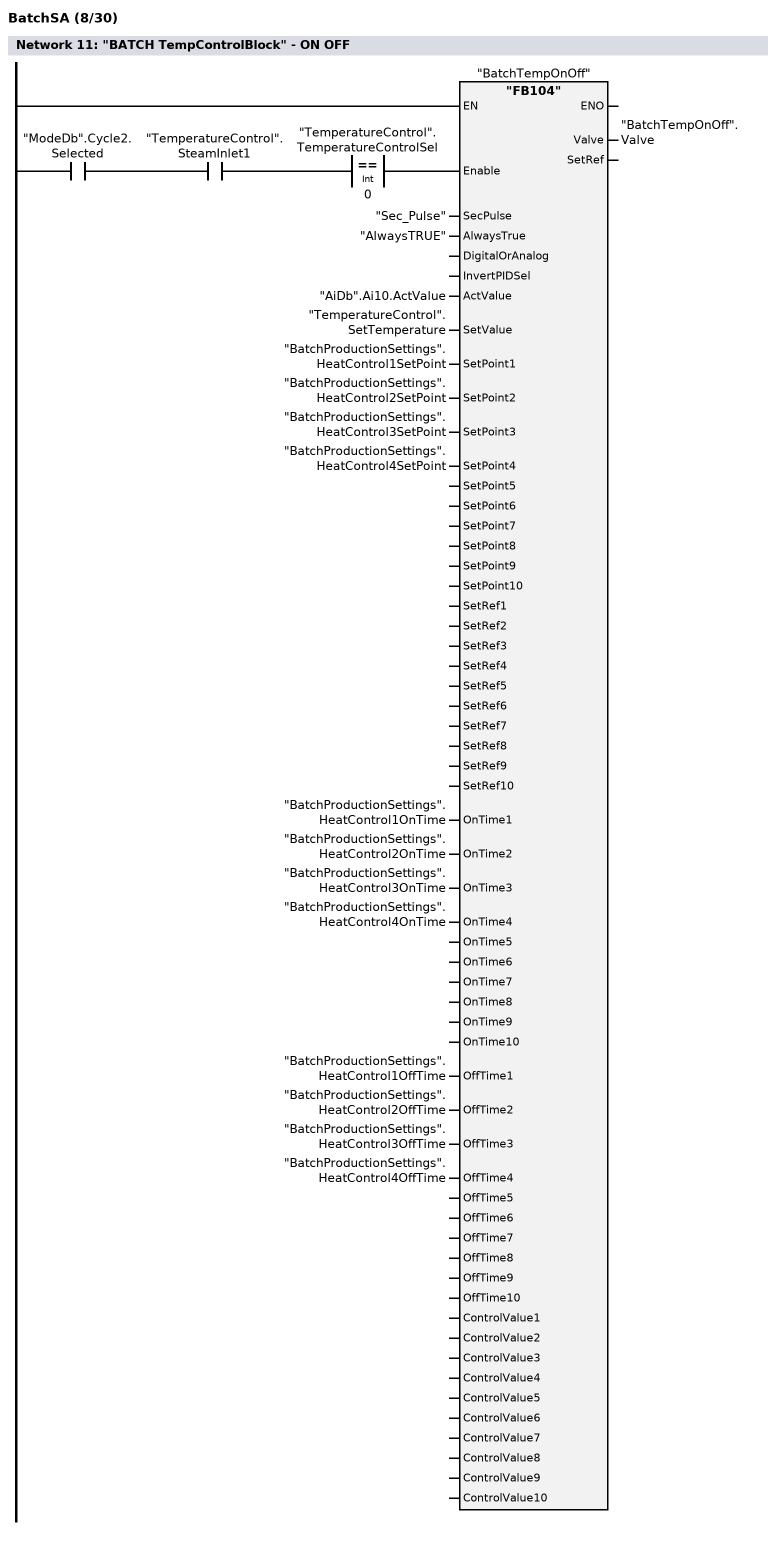
   RUNG wire#powerrail
      "BatchTempOnOff"(Enable := wire#w1, SecPulse := "Sec_Pulse", AlwaysTrue := "AlwaysTRUE", DigitalOrAnalog :=, InvertPIDSel :=, ActValue := "AiDb".Ai10.ActValue, SetValue := "TemperatureControl".SetTemperature, SetPoint1 := "BatchProductionSettings".HeatControl1SetPoint, SetPoint2 := "BatchProductionSettings".HeatControl2SetPoint, SetPoint3 := "BatchProductionSettings".HeatControl3SetPoint, SetPoint4 := "BatchProductionSettings".HeatControl4SetPoint, SetPoint5 :=, SetPoint6 :=, SetPoint7 :=, SetPoint8 :=, SetPoint9 :=, SetPoint10 :=, SetRef1 :=, SetRef2 :=, SetRef3 :=, SetRef4 :=, SetRef5 :=, SetRef6 :=, SetRef7 :=, SetRef8 :=, SetRef9 :=, SetRef10 :=, OnTime1 := "BatchProductionSettings".HeatControl1OnTime, OnTime2 := "BatchProductionSettings".HeatControl2OnTime, OnTime3 := "BatchProductionSettings".HeatControl3OnTime, OnTime4 := "BatchProductionSettings".HeatControl4OnTime, OnTime5 :=, OnTime6 :=, OnTime7 :=, OnTime8 :=, OnTime9 :=, OnTime10 :=, OffTime1 := "BatchProductionSettings".HeatControl1OffTime, OffTime2 := "BatchProductionSettings".HeatControl2OffTime, OffTime3 := "BatchProductionSettings".HeatControl3OffTime, OffTime4 := "BatchProductionSettings".HeatControl4OffTime, OffTime5 :=, OffTime6 :=, OffTime7 :=, OffTime8 :=, OffTime9 :=, OffTime10 :=, ControlValue1 :=, ControlValue2 :=, ControlValue3 :=, ControlValue4 :=, ControlValue5 :=, ControlValue6 :=, ControlValue7 :=, ControlValue8 :=, ControlValue9 :=, ControlValue10 :=, Valve => "BatchTempOnOff".Valve, SetRef =>)
   END_RUNG
   RUNG wire#powerrail
      Contact( "ModeDb".Cycle2.Selected )
      Contact( "TemperatureControl".SteamInlet1 )
      { S7_Templates := "SrcType := Int" } EQ_Contact(in1 := "TemperatureControl".TemperatureControlSel, in2 := 0)
   END_RUNG wire#w1
   // the same network as SCL:
   "BatchTempOnOff"(Enable := "ModeDb".Cycle2.Selected AND "TemperatureControl".SteamInlet1 AND ("TemperatureControl".TemperatureControlSel = 0),   // "FB104"
                    SecPulse := "Sec_Pulse",
                    AlwaysTrue := "AlwaysTRUE",
                    ActValue := "AiDb".Ai10.ActValue,
                    SetValue := "TemperatureControl".SetTemperature,
                    SetPoint1 := "BatchProductionSettings".HeatControl1SetPoint,
                    SetPoint2 := "BatchProductionSettings".HeatControl2SetPoint,
                    SetPoint3 := "BatchProductionSettings".HeatControl3SetPoint,
                    SetPoint4 := "BatchProductionSettings".HeatControl4SetPoint,
                    OnTime1 := "BatchProductionSettings".HeatControl1OnTime,
                    OnTime2 := "BatchProductionSettings".HeatControl2OnTime,
                    OnTime3 := "BatchProductionSettings".HeatControl3OnTime,
                    OnTime4 := "BatchProductionSettings".HeatControl4OnTime,
                    OffTime1 := "BatchProductionSettings".HeatControl1OffTime,
                    OffTime2 := "BatchProductionSettings".HeatControl2OffTime,
                    OffTime3 := "BatchProductionSettings".HeatControl3OffTime,
                    OffTime4 := "BatchProductionSettings".HeatControl4OffTime,
                    Valve => "BatchTempOnOff".Valve);
END_REGION

REGION Network 12: ******************************MM01 Mixing******************************
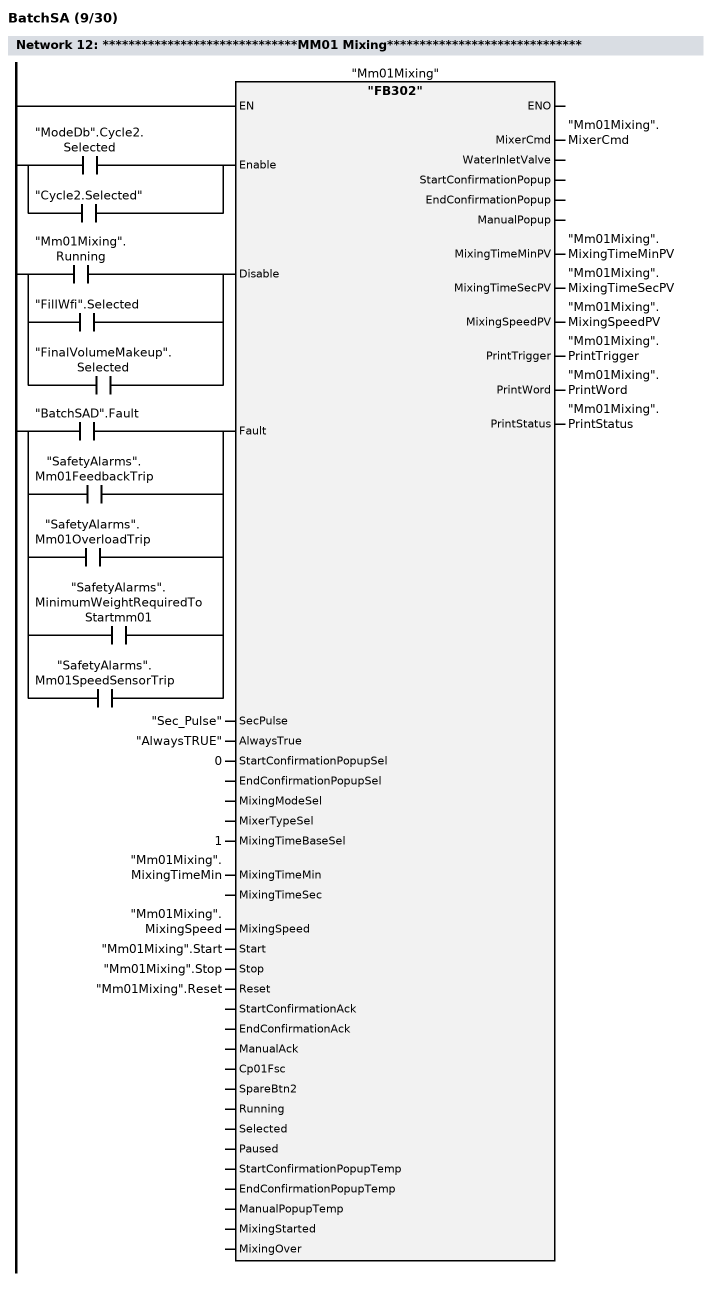
   RUNG wire#powerrail
      "Mm01Mixing"(Enable := wire#w1, Disable := wire#w2, Fault := wire#w3, SecPulse := "Sec_Pulse", AlwaysTrue := "AlwaysTRUE", StartConfirmationPopupSel := 0, EndConfirmationPopupSel :=, MixingModeSel :=, MixerTypeSel :=, MixingTimeBaseSel := 1, MixingTimeMin := "Mm01Mixing".MixingTimeMin, MixingTimeSec :=, MixingSpeed := "Mm01Mixing".MixingSpeed, Start := "Mm01Mixing".Start, Stop := "Mm01Mixing".Stop, Reset := "Mm01Mixing".Reset, StartConfirmationAck :=, EndConfirmationAck :=, ManualAck :=, Cp01Fsc :=, SpareBtn2 :=, Running :=, Selected :=, Paused :=, StartConfirmationPopupTemp :=, EndConfirmationPopupTemp :=, ManualPopupTemp :=, MixingStarted :=, MixingOver :=, MixerCmd => "Mm01Mixing".MixerCmd, WaterInletValve =>, StartConfirmationPopup =>, EndConfirmationPopup =>, ManualPopup =>, MixingTimeMinPV => "Mm01Mixing".MixingTimeMinPV, MixingTimeSecPV => "Mm01Mixing".MixingTimeSecPV, MixingSpeedPV => "Mm01Mixing".MixingSpeedPV, PrintTrigger => "Mm01Mixing".PrintTrigger, PrintWord => "Mm01Mixing".PrintWord, PrintStatus => "Mm01Mixing".PrintStatus)
   END_RUNG
   RUNG wire#powerrail
      Contact( "ModeDb".Cycle2.Selected )
   END_RUNG wire#w1
   RUNG wire#powerrail
      Contact( "Cycle2.Selected" )
   END_RUNG wire#w1
   RUNG wire#powerrail
      Contact( "Mm01Mixing".Running )
   END_RUNG wire#w2
   RUNG wire#powerrail
      Contact( "FillWfi".Selected )
   END_RUNG wire#w2
   RUNG wire#powerrail
      Contact( "FinalVolumeMakeup".Selected )
   END_RUNG wire#w2
   RUNG wire#powerrail
      Contact( "BatchSAD".Fault )
   END_RUNG wire#w3
   RUNG wire#powerrail
      Contact( "SafetyAlarms".Mm01FeedbackTrip )
   END_RUNG wire#w3
   RUNG wire#powerrail
      Contact( "SafetyAlarms".Mm01OverloadTrip )
   END_RUNG wire#w3
   RUNG wire#powerrail
      Contact( "SafetyAlarms".MinimumWeightRequiredToStartmm01 )
   END_RUNG wire#w3
   RUNG wire#powerrail
      Contact( "SafetyAlarms".Mm01SpeedSensorTrip )
   END_RUNG wire#w3
   // the same network as SCL:
   "Mm01Mixing"(Enable := "ModeDb".Cycle2.Selected OR "Cycle2.Selected",   // "FB302"
                Disable := "Mm01Mixing".Running OR "FillWfi".Selected OR "FinalVolumeMakeup".Selected,
                Fault := "BatchSAD".Fault OR "SafetyAlarms".Mm01FeedbackTrip OR "SafetyAlarms".Mm01OverloadTrip OR "SafetyAlarms".MinimumWeightRequiredToStartmm01 OR "SafetyAlarms".Mm01SpeedSensorTrip,
                SecPulse := "Sec_Pulse",
                AlwaysTrue := "AlwaysTRUE",
                StartConfirmationPopupSel := 0,
                MixingTimeBaseSel := 1,
                MixingTimeMin := "Mm01Mixing".MixingTimeMin,
                MixingSpeed := "Mm01Mixing".MixingSpeed,
                Start := "Mm01Mixing".Start,
                Stop := "Mm01Mixing".Stop,
                Reset := "Mm01Mixing".Reset,
                MixerCmd => "Mm01Mixing".MixerCmd,
                MixingTimeMinPV => "Mm01Mixing".MixingTimeMinPV,
                MixingTimeSecPV => "Mm01Mixing".MixingTimeSecPV,
                MixingSpeedPV => "Mm01Mixing".MixingSpeedPV,
                PrintTrigger => "Mm01Mixing".PrintTrigger,
                PrintWord => "Mm01Mixing".PrintWord,
                PrintStatus => "Mm01Mixing".PrintStatus);
END_REGION

REGION Network 13: Mm01 Mixing Event Staus
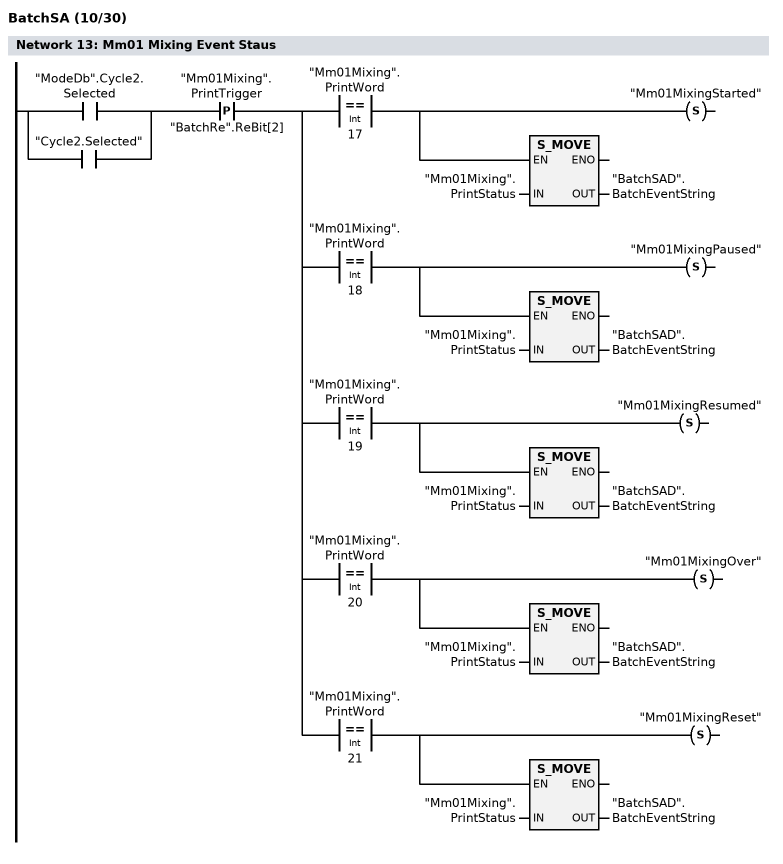
   RUNG wire#powerrail
      Contact( "ModeDb".Cycle2.Selected )
      wire#w1
      P_Contact(operand := "Mm01Mixing".PrintTrigger, bit := "BatchRe".ReBit[2])
      wire#w2
      { S7_Templates := "SrcType := Int" } EQ_Contact(in1 := "Mm01Mixing".PrintWord, in2 := 17)
      wire#w3
      S_Coil( "Mm01MixingStarted" )
   END_RUNG
   RUNG wire#powerrail
      Contact( "Cycle2.Selected" )
   END_RUNG wire#w1
   RUNG wire#w3
      S_Move(in := "Mm01Mixing".PrintStatus, out => "BatchSAD".BatchEventString)
   END_RUNG
   RUNG wire#w2
      { S7_Templates := "SrcType := Int" } EQ_Contact(in1 := "Mm01Mixing".PrintWord, in2 := 18)
      wire#w4
      S_Coil( "Mm01MixingPaused" )
   END_RUNG
   RUNG wire#w4
      S_Move(in := "Mm01Mixing".PrintStatus, out => "BatchSAD".BatchEventString)
   END_RUNG
   RUNG wire#w2
      { S7_Templates := "SrcType := Int" } EQ_Contact(in1 := "Mm01Mixing".PrintWord, in2 := 19)
      wire#w5
      S_Coil( "Mm01MixingResumed" )
   END_RUNG
   RUNG wire#w5
      S_Move(in := "Mm01Mixing".PrintStatus, out => "BatchSAD".BatchEventString)
   END_RUNG
   RUNG wire#w2
      { S7_Templates := "SrcType := Int" } EQ_Contact(in1 := "Mm01Mixing".PrintWord, in2 := 20)
      wire#w6
      S_Coil( "Mm01MixingOver" )
   END_RUNG
   RUNG wire#w6
      S_Move(in := "Mm01Mixing".PrintStatus, out => "BatchSAD".BatchEventString)
   END_RUNG
   RUNG wire#w2
      { S7_Templates := "SrcType := Int" } EQ_Contact(in1 := "Mm01Mixing".PrintWord, in2 := 21)
      wire#w7
      S_Coil( "Mm01MixingReset" )
   END_RUNG
   RUNG wire#w7
      S_Move(in := "Mm01Mixing".PrintStatus, out => "BatchSAD".BatchEventString)
   END_RUNG
   // the same network as SCL:
   #_w1 := ("ModeDb".Cycle2.Selected OR "Cycle2.Selected") AND "Mm01Mixing".PrintTrigger AND NOT "BatchRe".ReBit[2];   // rising edge of "Mm01Mixing".PrintTrigger
   "BatchRe".ReBit[2] := "Mm01Mixing".PrintTrigger;
   IF #_w1 AND ("Mm01Mixing".PrintWord = 17) THEN
       "Mm01MixingStarted" := TRUE;
       "BatchSAD".BatchEventString := "Mm01Mixing".PrintStatus;
   END_IF;
   IF #_w1 AND ("Mm01Mixing".PrintWord = 18) THEN
       "Mm01MixingPaused" := TRUE;
       "BatchSAD".BatchEventString := "Mm01Mixing".PrintStatus;
   END_IF;
   IF #_w1 AND ("Mm01Mixing".PrintWord = 19) THEN
       "Mm01MixingResumed" := TRUE;
       "BatchSAD".BatchEventString := "Mm01Mixing".PrintStatus;
   END_IF;
   IF #_w1 AND ("Mm01Mixing".PrintWord = 20) THEN
       "Mm01MixingOver" := TRUE;
       "BatchSAD".BatchEventString := "Mm01Mixing".PrintStatus;
   END_IF;
   IF #_w1 AND ("Mm01Mixing".PrintWord = 21) THEN
       "Mm01MixingReset" := TRUE;
       "BatchSAD".BatchEventString := "Mm01Mixing".PrintStatus;
   END_IF;
END_REGION

REGION Network 14: ******************************Rm Addition******************************
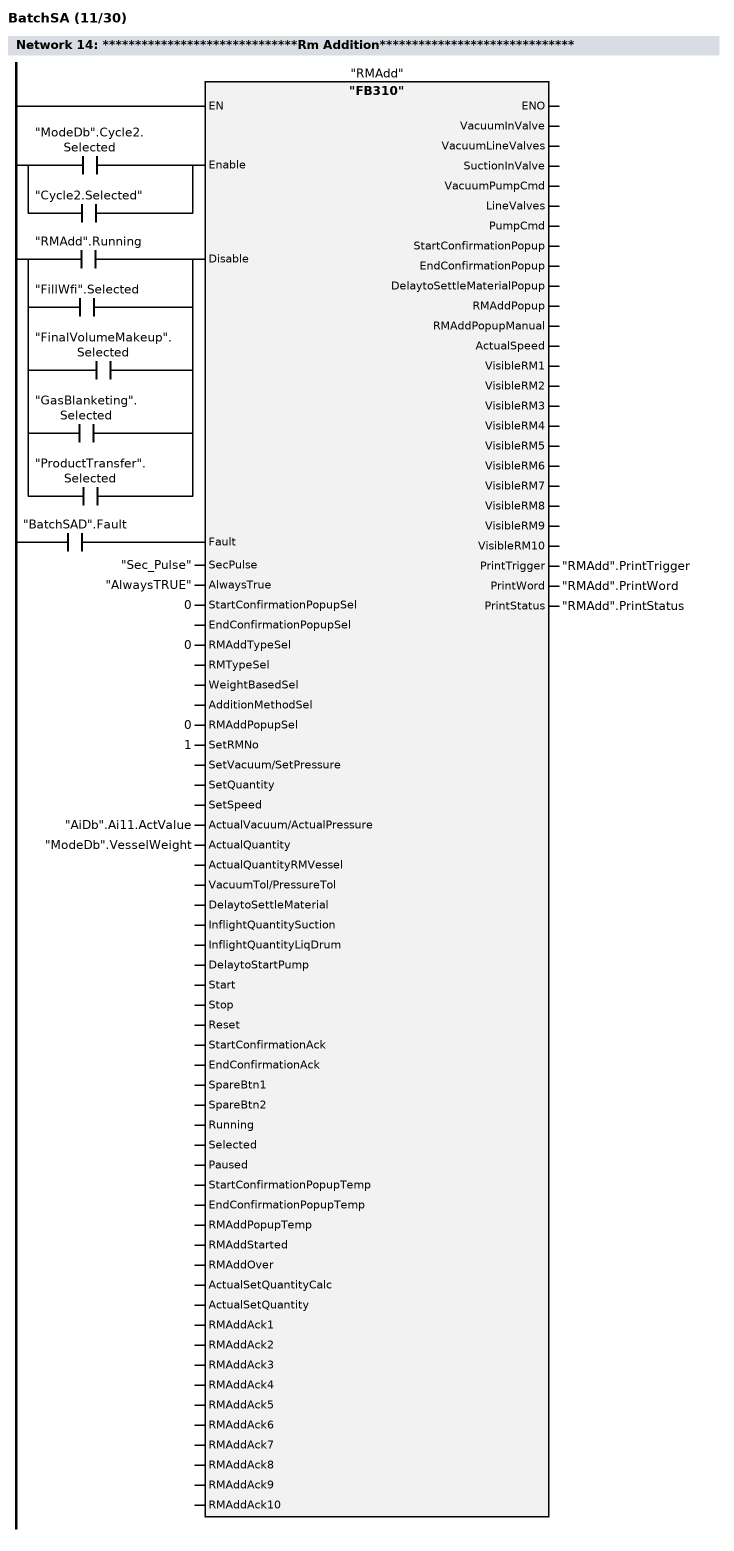
   RUNG wire#powerrail
      "RMAdd"(Enable := wire#w1, Disable := wire#w2, Fault := wire#w3, SecPulse := "Sec_Pulse", AlwaysTrue := "AlwaysTRUE", StartConfirmationPopupSel := 0, EndConfirmationPopupSel :=, RMAddTypeSel := 0, RMTypeSel :=, WeightBasedSel :=, AdditionMethodSel :=, RMAddPopupSel := 0, SetRMNo := 1, "SetVacuum/SetPressure" :=, SetQuantity :=, SetSpeed :=, "ActualVacuum/ActualPressure" := "AiDb".Ai11.ActValue, ActualQuantity := "ModeDb".VesselWeight, ActualQuantityRMVessel :=, "VacuumTol/PressureTol" :=, DelaytoSettleMaterial :=, InflightQuantitySuction :=, InflightQuantityLiqDrum :=, DelaytoStartPump :=, Start :=, Stop :=, Reset :=, StartConfirmationAck :=, EndConfirmationAck :=, SpareBtn1 :=, SpareBtn2 :=, Running :=, Selected :=, Paused :=, StartConfirmationPopupTemp :=, EndConfirmationPopupTemp :=, RMAddPopupTemp :=, RMAddStarted :=, RMAddOver :=, ActualSetQuantityCalc :=, ActualSetQuantity :=, RMAddAck1 :=, RMAddAck2 :=, RMAddAck3 :=, RMAddAck4 :=, RMAddAck5 :=, RMAddAck6 :=, RMAddAck7 :=, RMAddAck8 :=, RMAddAck9 :=, RMAddAck10 :=, VacuumInValve =>, VacuumLineValves =>, SuctionInValve =>, VacuumPumpCmd =>, LineValves =>, PumpCmd =>, StartConfirmationPopup =>, EndConfirmationPopup =>, DelaytoSettleMaterialPopup =>, RMAddPopup =>, RMAddPopupManual =>, ActualSpeed =>, VisibleRM1 =>, VisibleRM2 =>, VisibleRM3 =>, VisibleRM4 =>, VisibleRM5 =>, VisibleRM6 =>, VisibleRM7 =>, VisibleRM8 =>, VisibleRM9 =>, VisibleRM10 =>, PrintTrigger => "RMAdd".PrintTrigger, PrintWord => "RMAdd".PrintWord, PrintStatus => "RMAdd".PrintStatus)
   END_RUNG
   RUNG wire#powerrail
      Contact( "ModeDb".Cycle2.Selected )
   END_RUNG wire#w1
   RUNG wire#powerrail
      Contact( "Cycle2.Selected" )
   END_RUNG wire#w1
   RUNG wire#powerrail
      Contact( "RMAdd".Running )
   END_RUNG wire#w2
   RUNG wire#powerrail
      Contact( "FillWfi".Selected )
   END_RUNG wire#w2
   RUNG wire#powerrail
      Contact( "FinalVolumeMakeup".Selected )
   END_RUNG wire#w2
   RUNG wire#powerrail
      Contact( "GasBlanketing".Selected )
   END_RUNG wire#w2
   RUNG wire#powerrail
      Contact( "ProductTransfer".Selected )
   END_RUNG wire#w2
   RUNG wire#powerrail
      Contact( "BatchSAD".Fault )
   END_RUNG wire#w3
   // the same network as SCL:
   "RMAdd"(Enable := "ModeDb".Cycle2.Selected OR "Cycle2.Selected",   // "FB310"
           Disable := "RMAdd".Running OR "FillWfi".Selected OR "FinalVolumeMakeup".Selected OR "GasBlanketing".Selected OR "ProductTransfer".Selected,
           Fault := "BatchSAD".Fault,
           SecPulse := "Sec_Pulse",
           AlwaysTrue := "AlwaysTRUE",
           StartConfirmationPopupSel := 0,
           RMAddTypeSel := 0,
           RMAddPopupSel := 0,
           SetRMNo := 1,
           "ActualVacuum/ActualPressure" := "AiDb".Ai11.ActValue,
           ActualQuantity := "ModeDb".VesselWeight,
           PrintTrigger => "RMAdd".PrintTrigger,
           PrintWord => "RMAdd".PrintWord,
           PrintStatus => "RMAdd".PrintStatus);
END_REGION

REGION Network 15: "BatchSAD".RmAddVesselSafetyPressurePopup
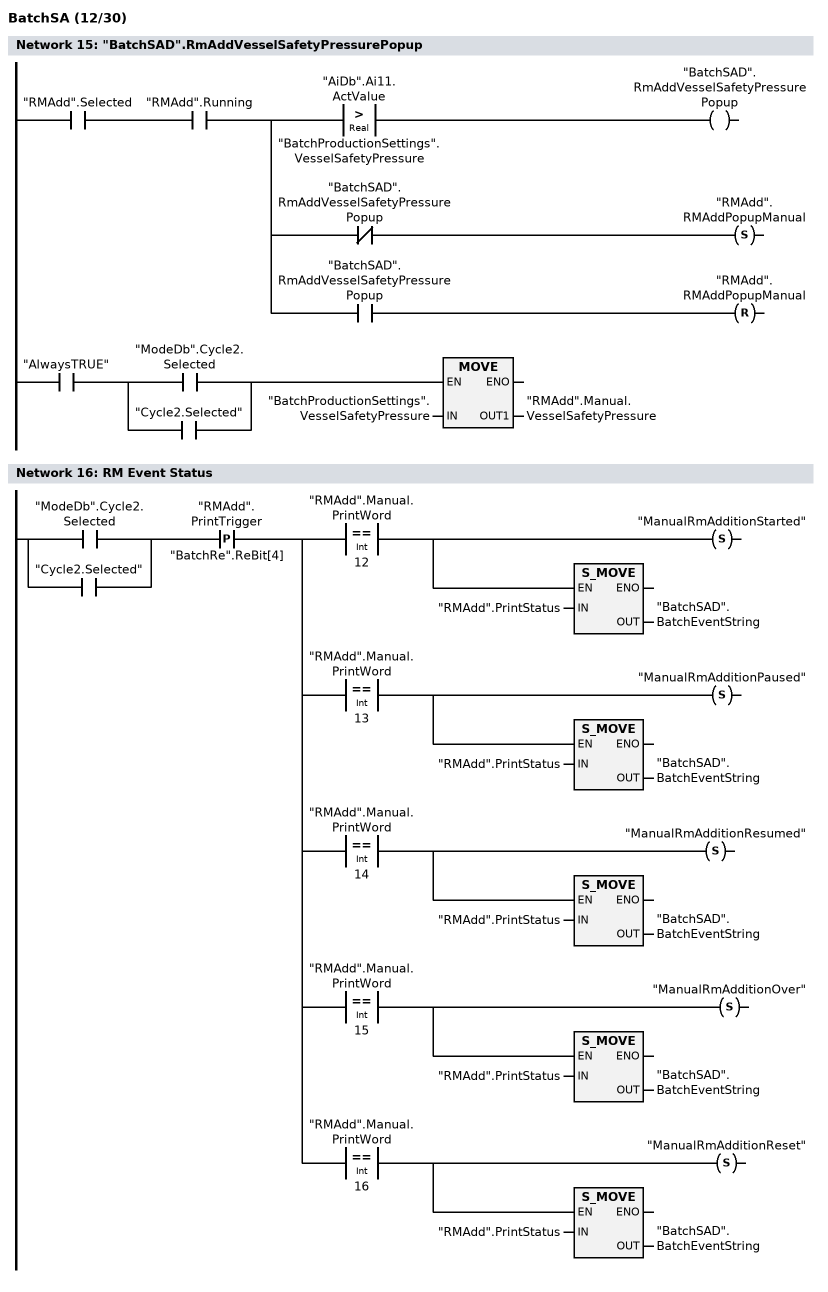
   RUNG wire#powerrail
      Contact( "RMAdd".Selected )
      Contact( "RMAdd".Running )
      wire#w1
      { S7_Templates := "SrcType := Real" } GT_Contact(in1 := "AiDb".Ai11.ActValue, in2 := "BatchProductionSettings".VesselSafetyPressure)
      Coil( "BatchSAD".RmAddVesselSafetyPressurePopup )
   END_RUNG
   RUNG wire#w1
      I_Contact( "BatchSAD".RmAddVesselSafetyPressurePopup )
      S_Coil( "RMAdd".RMAddPopupManual )
   END_RUNG
   RUNG wire#w1
      Contact( "BatchSAD".RmAddVesselSafetyPressurePopup )
      R_Coil( "RMAdd".RMAddPopupManual )
   END_RUNG
   RUNG wire#powerrail
      Contact( "AlwaysTRUE" )
      wire#w2
      Contact( "ModeDb".Cycle2.Selected )
      wire#w3
      Move(in := "BatchProductionSettings".VesselSafetyPressure, out1 => "RMAdd".Manual.VesselSafetyPressure)
   END_RUNG
   RUNG wire#w2
      Contact( "Cycle2.Selected" )
   END_RUNG wire#w3
   // the same network as SCL:
   #_w1 := "RMAdd".Selected AND "RMAdd".Running;
   "BatchSAD".RmAddVesselSafetyPressurePopup := #_w1 AND ("AiDb".Ai11.ActValue > "BatchProductionSettings".VesselSafetyPressure);
   IF #_w1 AND NOT "BatchSAD".RmAddVesselSafetyPressurePopup THEN "RMAdd".RMAddPopupManual := TRUE; END_IF;
   IF #_w1 AND "BatchSAD".RmAddVesselSafetyPressurePopup THEN "RMAdd".RMAddPopupManual := FALSE; END_IF;
   IF "AlwaysTRUE" AND ("ModeDb".Cycle2.Selected OR "Cycle2.Selected") THEN
       "RMAdd".Manual.VesselSafetyPressure := "BatchProductionSettings".VesselSafetyPressure;
   END_IF;
END_REGION

REGION Network 16: RM Event Status
   RUNG wire#powerrail
      Contact( "ModeDb".Cycle2.Selected )
      wire#w1
      P_Contact(operand := "RMAdd".PrintTrigger, bit := "BatchRe".ReBit[4])
      wire#w2
      { S7_Templates := "SrcType := Int" } EQ_Contact(in1 := "RMAdd".Manual.PrintWord, in2 := 12)
      wire#w3
      S_Coil( "ManualRmAdditionStarted" )
   END_RUNG
   RUNG wire#powerrail
      Contact( "Cycle2.Selected" )
   END_RUNG wire#w1
   RUNG wire#w3
      S_Move(in := "RMAdd".PrintStatus, out => "BatchSAD".BatchEventString)
   END_RUNG
   RUNG wire#w2
      { S7_Templates := "SrcType := Int" } EQ_Contact(in1 := "RMAdd".Manual.PrintWord, in2 := 13)
      wire#w4
      S_Coil( "ManualRmAdditionPaused" )
   END_RUNG
   RUNG wire#w4
      S_Move(in := "RMAdd".PrintStatus, out => "BatchSAD".BatchEventString)
   END_RUNG
   RUNG wire#w2
      { S7_Templates := "SrcType := Int" } EQ_Contact(in1 := "RMAdd".Manual.PrintWord, in2 := 14)
      wire#w5
      S_Coil( "ManualRmAdditionResumed" )
   END_RUNG
   RUNG wire#w5
      S_Move(in := "RMAdd".PrintStatus, out => "BatchSAD".BatchEventString)
   END_RUNG
   RUNG wire#w2
      { S7_Templates := "SrcType := Int" } EQ_Contact(in1 := "RMAdd".Manual.PrintWord, in2 := 15)
      wire#w6
      S_Coil( "ManualRmAdditionOver" )
   END_RUNG
   RUNG wire#w6
      S_Move(in := "RMAdd".PrintStatus, out => "BatchSAD".BatchEventString)
   END_RUNG
   RUNG wire#w2
      { S7_Templates := "SrcType := Int" } EQ_Contact(in1 := "RMAdd".Manual.PrintWord, in2 := 16)
      wire#w7
      S_Coil( "ManualRmAdditionReset" )
   END_RUNG
   RUNG wire#w7
      S_Move(in := "RMAdd".PrintStatus, out => "BatchSAD".BatchEventString)
   END_RUNG
   // the same network as SCL:
   #_w1 := ("ModeDb".Cycle2.Selected OR "Cycle2.Selected") AND "RMAdd".PrintTrigger AND NOT "BatchRe".ReBit[4];   // rising edge of "RMAdd".PrintTrigger
   "BatchRe".ReBit[4] := "RMAdd".PrintTrigger;
   IF #_w1 AND ("RMAdd".Manual.PrintWord = 12) THEN
       "ManualRmAdditionStarted" := TRUE;
       "BatchSAD".BatchEventString := "RMAdd".PrintStatus;
   END_IF;
   IF #_w1 AND ("RMAdd".Manual.PrintWord = 13) THEN
       "ManualRmAdditionPaused" := TRUE;
       "BatchSAD".BatchEventString := "RMAdd".PrintStatus;
   END_IF;
   IF #_w1 AND ("RMAdd".Manual.PrintWord = 14) THEN
       "ManualRmAdditionResumed" := TRUE;
       "BatchSAD".BatchEventString := "RMAdd".PrintStatus;
   END_IF;
   IF #_w1 AND ("RMAdd".Manual.PrintWord = 15) THEN
       "ManualRmAdditionOver" := TRUE;
       "BatchSAD".BatchEventString := "RMAdd".PrintStatus;
   END_IF;
   IF #_w1 AND ("RMAdd".Manual.PrintWord = 16) THEN
       "ManualRmAdditionReset" := TRUE;
       "BatchSAD".BatchEventString := "RMAdd".PrintStatus;
   END_IF;
END_REGION

REGION Network 17: ******************************N2 Sparging******************************
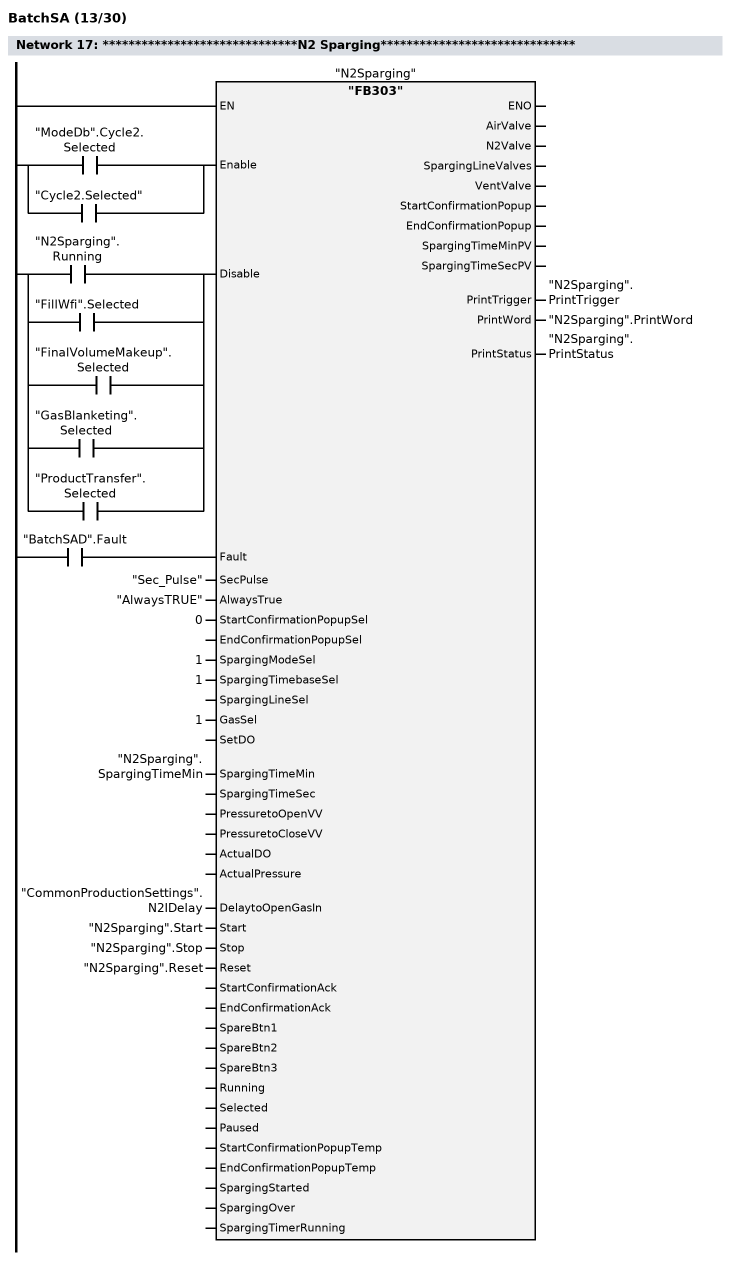
   RUNG wire#powerrail
      "N2Sparging"(Enable := wire#w1, Disable := wire#w2, Fault := wire#w3, SecPulse := "Sec_Pulse", AlwaysTrue := "AlwaysTRUE", StartConfirmationPopupSel := 0, EndConfirmationPopupSel :=, SpargingModeSel := 1, SpargingTimebaseSel := 1, SpargingLineSel :=, GasSel := 1, SetDO :=, SpargingTimeMin := "N2Sparging".SpargingTimeMin, SpargingTimeSec :=, PressuretoOpenVV :=, PressuretoCloseVV :=, ActualDO :=, ActualPressure :=, DelaytoOpenGasIn := "CommonProductionSettings".N2IDelay, Start := "N2Sparging".Start, Stop := "N2Sparging".Stop, Reset := "N2Sparging".Reset, StartConfirmationAck :=, EndConfirmationAck :=, SpareBtn1 :=, SpareBtn2 :=, SpareBtn3 :=, Running :=, Selected :=, Paused :=, StartConfirmationPopupTemp :=, EndConfirmationPopupTemp :=, SpargingStarted :=, SpargingOver :=, SpargingTimerRunning :=, AirValve =>, N2Valve =>, SpargingLineValves =>, VentValve =>, StartConfirmationPopup =>, EndConfirmationPopup =>, SpargingTimeMinPV =>, SpargingTimeSecPV =>, PrintTrigger => "N2Sparging".PrintTrigger, PrintWord => "N2Sparging".PrintWord, PrintStatus => "N2Sparging".PrintStatus)
   END_RUNG
   RUNG wire#powerrail
      Contact( "ModeDb".Cycle2.Selected )
   END_RUNG wire#w1
   RUNG wire#powerrail
      Contact( "Cycle2.Selected" )
   END_RUNG wire#w1
   RUNG wire#powerrail
      Contact( "N2Sparging".Running )
   END_RUNG wire#w2
   RUNG wire#powerrail
      Contact( "FillWfi".Selected )
   END_RUNG wire#w2
   RUNG wire#powerrail
      Contact( "FinalVolumeMakeup".Selected )
   END_RUNG wire#w2
   RUNG wire#powerrail
      Contact( "GasBlanketing".Selected )
   END_RUNG wire#w2
   RUNG wire#powerrail
      Contact( "ProductTransfer".Selected )
   END_RUNG wire#w2
   RUNG wire#powerrail
      Contact( "BatchSAD".Fault )
   END_RUNG wire#w3
   // the same network as SCL:
   "N2Sparging"(Enable := "ModeDb".Cycle2.Selected OR "Cycle2.Selected",   // "FB303"
                Disable := "N2Sparging".Running OR "FillWfi".Selected OR "FinalVolumeMakeup".Selected OR "GasBlanketing".Selected OR "ProductTransfer".Selected,
                Fault := "BatchSAD".Fault,
                SecPulse := "Sec_Pulse",
                AlwaysTrue := "AlwaysTRUE",
                StartConfirmationPopupSel := 0,
                SpargingModeSel := 1,
                SpargingTimebaseSel := 1,
                GasSel := 1,
                SpargingTimeMin := "N2Sparging".SpargingTimeMin,
                DelaytoOpenGasIn := "CommonProductionSettings".N2IDelay,
                Start := "N2Sparging".Start,
                Stop := "N2Sparging".Stop,
                Reset := "N2Sparging".Reset,
                PrintTrigger => "N2Sparging".PrintTrigger,
                PrintWord => "N2Sparging".PrintWord,
                PrintStatus => "N2Sparging".PrintStatus);
END_REGION

REGION Network 18: N2 Sparging Event Status
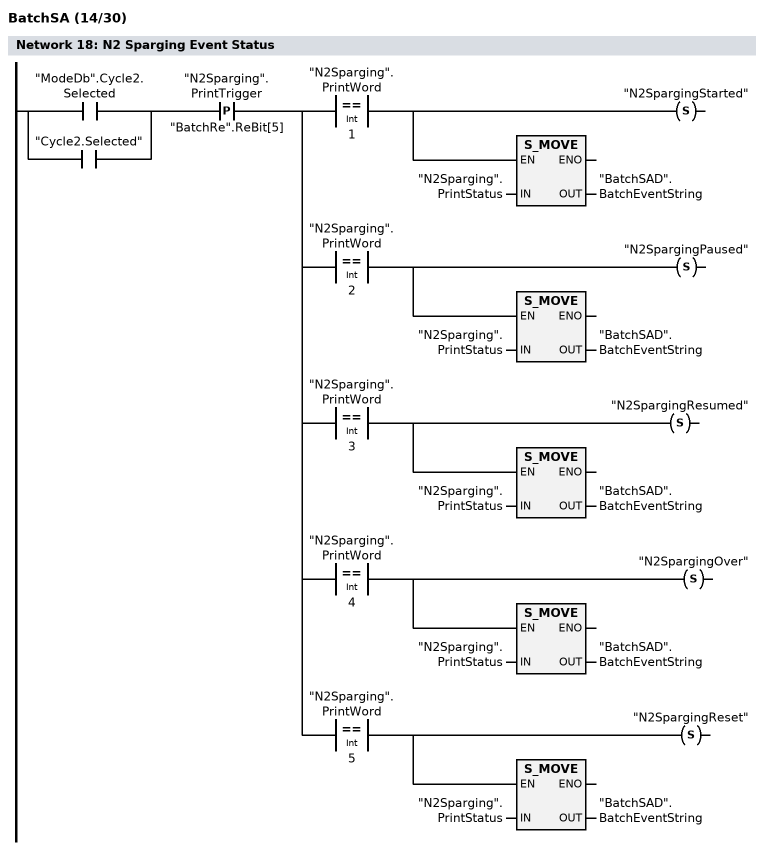
   RUNG wire#powerrail
      Contact( "ModeDb".Cycle2.Selected )
      wire#w1
      P_Contact(operand := "N2Sparging".PrintTrigger, bit := "BatchRe".ReBit[5])
      wire#w2
      { S7_Templates := "SrcType := Int" } EQ_Contact(in1 := "N2Sparging".PrintWord, in2 := 1)
      wire#w3
      S_Coil( "N2SpargingStarted" )
   END_RUNG
   RUNG wire#powerrail
      Contact( "Cycle2.Selected" )
   END_RUNG wire#w1
   RUNG wire#w3
      S_Move(in := "N2Sparging".PrintStatus, out => "BatchSAD".BatchEventString)
   END_RUNG
   RUNG wire#w2
      { S7_Templates := "SrcType := Int" } EQ_Contact(in1 := "N2Sparging".PrintWord, in2 := 2)
      wire#w4
      S_Coil( "N2SpargingPaused" )
   END_RUNG
   RUNG wire#w4
      S_Move(in := "N2Sparging".PrintStatus, out => "BatchSAD".BatchEventString)
   END_RUNG
   RUNG wire#w2
      { S7_Templates := "SrcType := Int" } EQ_Contact(in1 := "N2Sparging".PrintWord, in2 := 3)
      wire#w5
      S_Coil( "N2SpargingResumed" )
   END_RUNG
   RUNG wire#w5
      S_Move(in := "N2Sparging".PrintStatus, out => "BatchSAD".BatchEventString)
   END_RUNG
   RUNG wire#w2
      { S7_Templates := "SrcType := Int" } EQ_Contact(in1 := "N2Sparging".PrintWord, in2 := 4)
      wire#w6
      S_Coil( "N2SpargingOver" )
   END_RUNG
   RUNG wire#w6
      S_Move(in := "N2Sparging".PrintStatus, out => "BatchSAD".BatchEventString)
   END_RUNG
   RUNG wire#w2
      { S7_Templates := "SrcType := Int" } EQ_Contact(in1 := "N2Sparging".PrintWord, in2 := 5)
      wire#w7
      S_Coil( "N2SpargingReset" )
   END_RUNG
   RUNG wire#w7
      S_Move(in := "N2Sparging".PrintStatus, out => "BatchSAD".BatchEventString)
   END_RUNG
   // the same network as SCL:
   #_w1 := ("ModeDb".Cycle2.Selected OR "Cycle2.Selected") AND "N2Sparging".PrintTrigger AND NOT "BatchRe".ReBit[5];   // rising edge of "N2Sparging".PrintTrigger
   "BatchRe".ReBit[5] := "N2Sparging".PrintTrigger;
   IF #_w1 AND ("N2Sparging".PrintWord = 1) THEN
       "N2SpargingStarted" := TRUE;
       "BatchSAD".BatchEventString := "N2Sparging".PrintStatus;
   END_IF;
   IF #_w1 AND ("N2Sparging".PrintWord = 2) THEN
       "N2SpargingPaused" := TRUE;
       "BatchSAD".BatchEventString := "N2Sparging".PrintStatus;
   END_IF;
   IF #_w1 AND ("N2Sparging".PrintWord = 3) THEN
       "N2SpargingResumed" := TRUE;
       "BatchSAD".BatchEventString := "N2Sparging".PrintStatus;
   END_IF;
   IF #_w1 AND ("N2Sparging".PrintWord = 4) THEN
       "N2SpargingOver" := TRUE;
       "BatchSAD".BatchEventString := "N2Sparging".PrintStatus;
   END_IF;
   IF #_w1 AND ("N2Sparging".PrintWord = 5) THEN
       "N2SpargingReset" := TRUE;
       "BatchSAD".BatchEventString := "N2Sparging".PrintStatus;
   END_IF;
END_REGION

REGION Network 19: ******************************GasBlanketing******************************
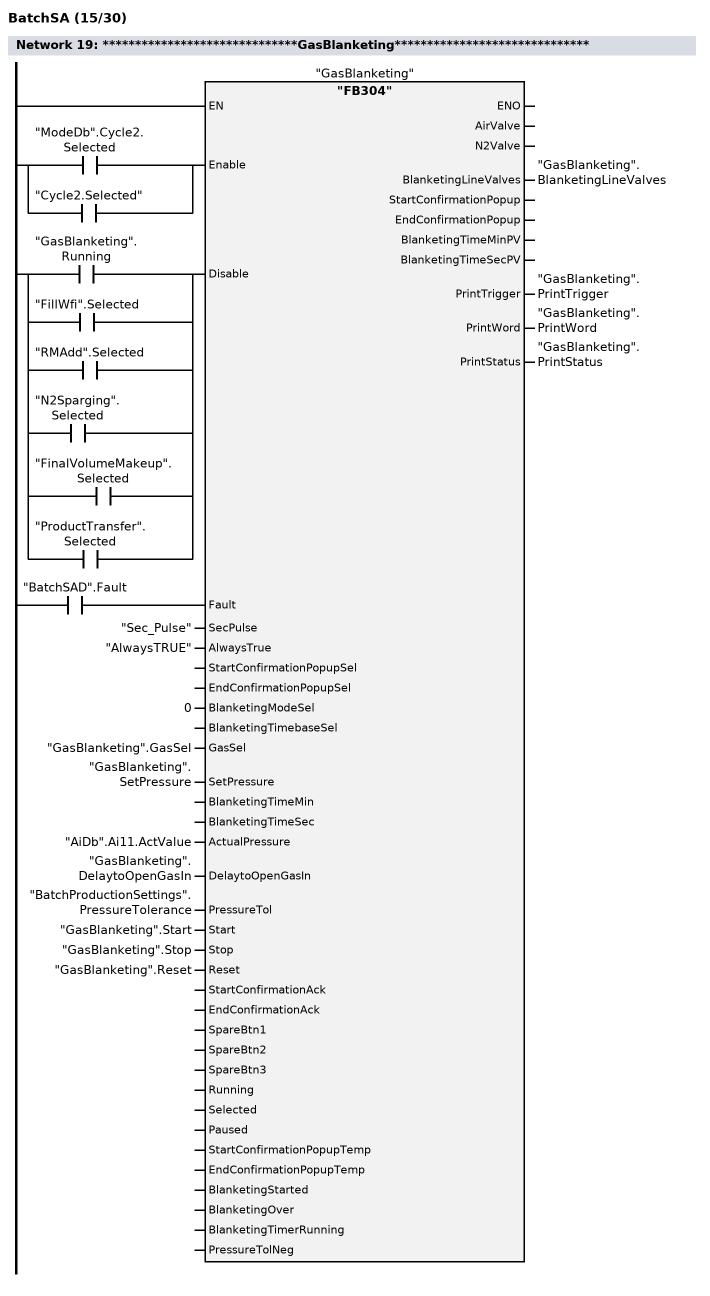
   RUNG wire#powerrail
      "GasBlanketing"(Enable := wire#w1, Disable := wire#w2, Fault := wire#w3, SecPulse := "Sec_Pulse", AlwaysTrue := "AlwaysTRUE", StartConfirmationPopupSel :=, EndConfirmationPopupSel :=, BlanketingModeSel := 0, BlanketingTimebaseSel :=, GasSel := "GasBlanketing".GasSel, SetPressure := "GasBlanketing".SetPressure, BlanketingTimeMin :=, BlanketingTimeSec :=, ActualPressure := "AiDb".Ai11.ActValue, DelaytoOpenGasIn := "GasBlanketing".DelaytoOpenGasIn, PressureTol := "BatchProductionSettings".PressureTolerance, Start := "GasBlanketing".Start, Stop := "GasBlanketing".Stop, Reset := "GasBlanketing".Reset, StartConfirmationAck :=, EndConfirmationAck :=, SpareBtn1 :=, SpareBtn2 :=, SpareBtn3 :=, Running :=, Selected :=, Paused :=, StartConfirmationPopupTemp :=, EndConfirmationPopupTemp :=, BlanketingStarted :=, BlanketingOver :=, BlanketingTimerRunning :=, PressureTolNeg :=, AirValve =>, N2Valve =>, BlanketingLineValves => "GasBlanketing".BlanketingLineValves, StartConfirmationPopup =>, EndConfirmationPopup =>, BlanketingTimeMinPV =>, BlanketingTimeSecPV =>, PrintTrigger => "GasBlanketing".PrintTrigger, PrintWord => "GasBlanketing".PrintWord, PrintStatus => "GasBlanketing".PrintStatus)
   END_RUNG
   RUNG wire#powerrail
      Contact( "ModeDb".Cycle2.Selected )
   END_RUNG wire#w1
   RUNG wire#powerrail
      Contact( "Cycle2.Selected" )
   END_RUNG wire#w1
   RUNG wire#powerrail
      Contact( "GasBlanketing".Running )
   END_RUNG wire#w2
   RUNG wire#powerrail
      Contact( "FillWfi".Selected )
   END_RUNG wire#w2
   RUNG wire#powerrail
      Contact( "RMAdd".Selected )
   END_RUNG wire#w2
   RUNG wire#powerrail
      Contact( "N2Sparging".Selected )
   END_RUNG wire#w2
   RUNG wire#powerrail
      Contact( "FinalVolumeMakeup".Selected )
   END_RUNG wire#w2
   RUNG wire#powerrail
      Contact( "ProductTransfer".Selected )
   END_RUNG wire#w2
   RUNG wire#powerrail
      Contact( "BatchSAD".Fault )
   END_RUNG wire#w3
   // the same network as SCL:
   "GasBlanketing"(Enable := "ModeDb".Cycle2.Selected OR "Cycle2.Selected",   // "FB304"
                   Disable := "GasBlanketing".Running OR "FillWfi".Selected OR "RMAdd".Selected OR "N2Sparging".Selected OR "FinalVolumeMakeup".Selected OR "ProductTransfer".Selected,
                   Fault := "BatchSAD".Fault,
                   SecPulse := "Sec_Pulse",
                   AlwaysTrue := "AlwaysTRUE",
                   BlanketingModeSel := 0,
                   GasSel := "GasBlanketing".GasSel,
                   SetPressure := "GasBlanketing".SetPressure,
                   ActualPressure := "AiDb".Ai11.ActValue,
                   DelaytoOpenGasIn := "GasBlanketing".DelaytoOpenGasIn,
                   PressureTol := "BatchProductionSettings".PressureTolerance,
                   Start := "GasBlanketing".Start,
                   Stop := "GasBlanketing".Stop,
                   Reset := "GasBlanketing".Reset,
                   BlanketingLineValves => "GasBlanketing".BlanketingLineValves,
                   PrintTrigger => "GasBlanketing".PrintTrigger,
                   PrintWord => "GasBlanketing".PrintWord,
                   PrintStatus => "GasBlanketing".PrintStatus);
END_REGION

REGION Network 20: GasBlanketing Event Status
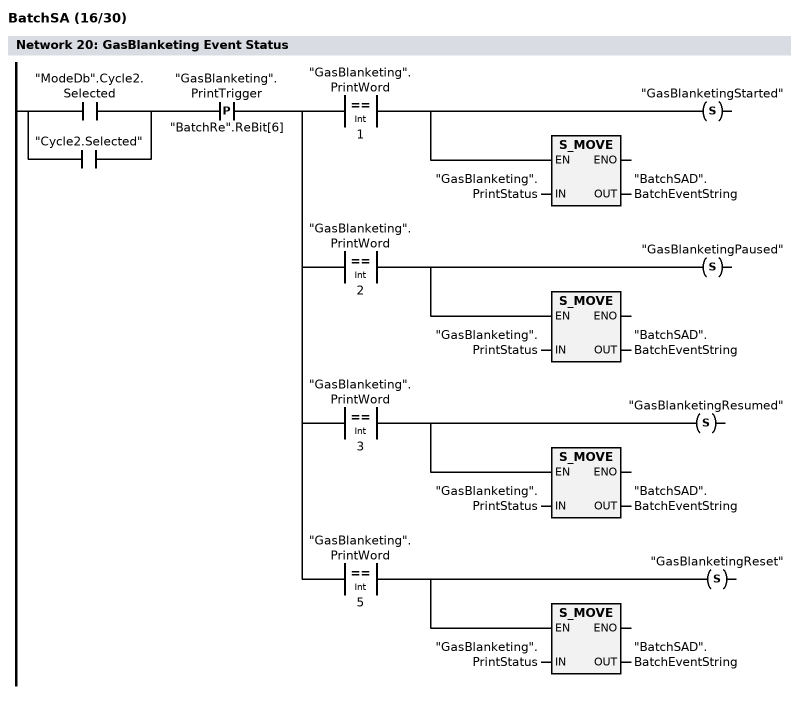
   RUNG wire#powerrail
      Contact( "ModeDb".Cycle2.Selected )
      wire#w1
      P_Contact(operand := "GasBlanketing".PrintTrigger, bit := "BatchRe".ReBit[6])
      wire#w2
      { S7_Templates := "SrcType := Int" } EQ_Contact(in1 := "GasBlanketing".PrintWord, in2 := 1)
      wire#w3
      S_Coil( "GasBlanketingStarted" )
   END_RUNG
   RUNG wire#powerrail
      Contact( "Cycle2.Selected" )
   END_RUNG wire#w1
   RUNG wire#w3
      S_Move(in := "GasBlanketing".PrintStatus, out => "BatchSAD".BatchEventString)
   END_RUNG
   RUNG wire#w2
      { S7_Templates := "SrcType := Int" } EQ_Contact(in1 := "GasBlanketing".PrintWord, in2 := 2)
      wire#w4
      S_Coil( "GasBlanketingPaused" )
   END_RUNG
   RUNG wire#w4
      S_Move(in := "GasBlanketing".PrintStatus, out => "BatchSAD".BatchEventString)
   END_RUNG
   RUNG wire#w2
      { S7_Templates := "SrcType := Int" } EQ_Contact(in1 := "GasBlanketing".PrintWord, in2 := 3)
      wire#w5
      S_Coil( "GasBlanketingResumed" )
   END_RUNG
   RUNG wire#w5
      S_Move(in := "GasBlanketing".PrintStatus, out => "BatchSAD".BatchEventString)
   END_RUNG
   RUNG wire#w2
      { S7_Templates := "SrcType := Int" } EQ_Contact(in1 := "GasBlanketing".PrintWord, in2 := 5)
      wire#w6
      S_Coil( "GasBlanketingReset" )
   END_RUNG
   RUNG wire#w6
      S_Move(in := "GasBlanketing".PrintStatus, out => "BatchSAD".BatchEventString)
   END_RUNG
   // the same network as SCL:
   #_w1 := ("ModeDb".Cycle2.Selected OR "Cycle2.Selected") AND "GasBlanketing".PrintTrigger AND NOT "BatchRe".ReBit[6];   // rising edge of "GasBlanketing".PrintTrigger
   "BatchRe".ReBit[6] := "GasBlanketing".PrintTrigger;
   IF #_w1 AND ("GasBlanketing".PrintWord = 1) THEN
       "GasBlanketingStarted" := TRUE;
       "BatchSAD".BatchEventString := "GasBlanketing".PrintStatus;
   END_IF;
   IF #_w1 AND ("GasBlanketing".PrintWord = 2) THEN
       "GasBlanketingPaused" := TRUE;
       "BatchSAD".BatchEventString := "GasBlanketing".PrintStatus;
   END_IF;
   IF #_w1 AND ("GasBlanketing".PrintWord = 3) THEN
       "GasBlanketingResumed" := TRUE;
       "BatchSAD".BatchEventString := "GasBlanketing".PrintStatus;
   END_IF;
   IF #_w1 AND ("GasBlanketing".PrintWord = 5) THEN
       "GasBlanketingReset" := TRUE;
       "BatchSAD".BatchEventString := "GasBlanketing".PrintStatus;
   END_IF;
END_REGION

REGION Network 21: ******************************FinalVolumeMakeup******************************
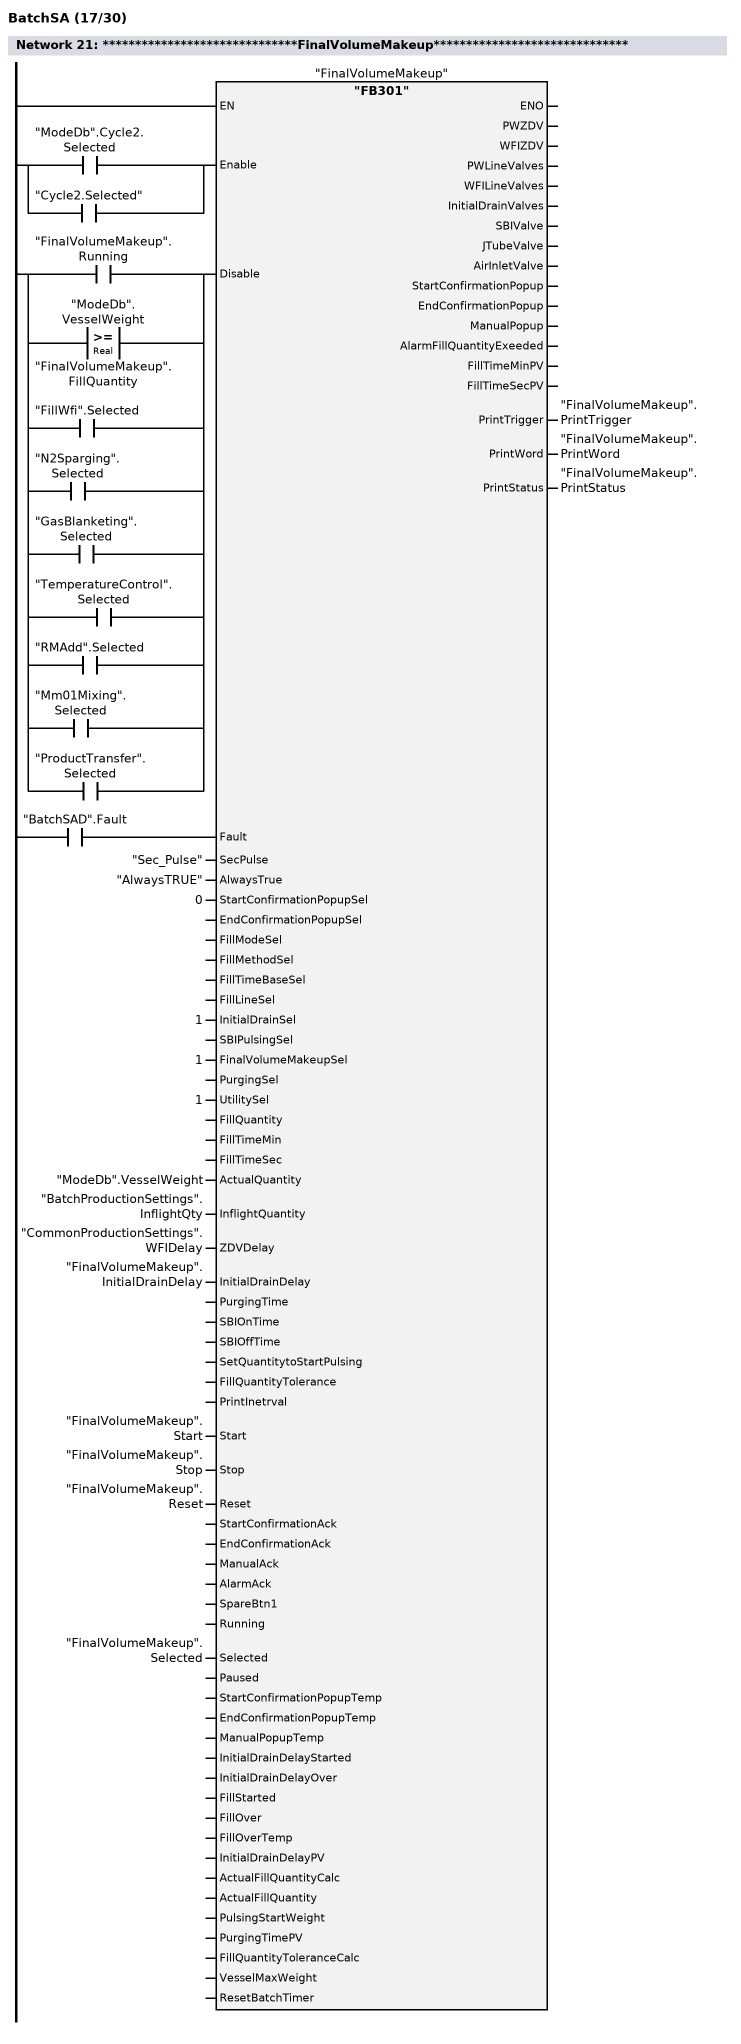
   RUNG wire#powerrail
      "FinalVolumeMakeup"(Enable := wire#w1, Disable := wire#w2, Fault := wire#w3, SecPulse := "Sec_Pulse", AlwaysTrue := "AlwaysTRUE", StartConfirmationPopupSel := 0, EndConfirmationPopupSel :=, FillModeSel :=, FillMethodSel :=, FillTimeBaseSel :=, FillLineSel :=, InitialDrainSel := 1, SBIPulsingSel :=, FinalVolumeMakeupSel := 1, PurgingSel :=, UtilitySel := 1, FillQuantity :=, FillTimeMin :=, FillTimeSec :=, ActualQuantity := "ModeDb".VesselWeight, InflightQuantity := "BatchProductionSettings".InflightQty, ZDVDelay := "CommonProductionSettings".WFIDelay, InitialDrainDelay := "FinalVolumeMakeup".InitialDrainDelay, PurgingTime :=, SBIOnTime :=, SBIOffTime :=, SetQuantitytoStartPulsing :=, FillQuantityTolerance :=, PrintInetrval :=, Start := "FinalVolumeMakeup".Start, Stop := "FinalVolumeMakeup".Stop, Reset := "FinalVolumeMakeup".Reset, StartConfirmationAck :=, EndConfirmationAck :=, ManualAck :=, AlarmAck :=, SpareBtn1 :=, Running :=, Selected := "FinalVolumeMakeup".Selected, Paused :=, StartConfirmationPopupTemp :=, EndConfirmationPopupTemp :=, ManualPopupTemp :=, InitialDrainDelayStarted :=, InitialDrainDelayOver :=, FillStarted :=, FillOver :=, FillOverTemp :=, InitialDrainDelayPV :=, ActualFillQuantityCalc :=, ActualFillQuantity :=, PulsingStartWeight :=, PurgingTimePV :=, FillQuantityToleranceCalc :=, VesselMaxWeight :=, ResetBatchTimer :=, PWZDV =>, WFIZDV =>, PWLineValves =>, WFILineValves =>, InitialDrainValves =>, SBIValve =>, JTubeValve =>, AirInletValve =>, StartConfirmationPopup =>, EndConfirmationPopup =>, ManualPopup =>, AlarmFillQuantityExeeded =>, FillTimeMinPV =>, FillTimeSecPV =>, PrintTrigger => "FinalVolumeMakeup".PrintTrigger, PrintWord => "FinalVolumeMakeup".PrintWord, PrintStatus => "FinalVolumeMakeup".PrintStatus)
   END_RUNG
   RUNG wire#powerrail
      Contact( "ModeDb".Cycle2.Selected )
   END_RUNG wire#w1
   RUNG wire#powerrail
      Contact( "Cycle2.Selected" )
   END_RUNG wire#w1
   RUNG wire#powerrail
      Contact( "FinalVolumeMakeup".Running )
   END_RUNG wire#w2
   RUNG wire#powerrail
      { S7_Templates := "SrcType := Real" } GE_Contact(in1 := "ModeDb".VesselWeight, in2 := "FinalVolumeMakeup".FillQuantity)
   END_RUNG wire#w2
   RUNG wire#powerrail
      Contact( "FillWfi".Selected )
   END_RUNG wire#w2
   RUNG wire#powerrail
      Contact( "N2Sparging".Selected )
   END_RUNG wire#w2
   RUNG wire#powerrail
      Contact( "GasBlanketing".Selected )
   END_RUNG wire#w2
   RUNG wire#powerrail
      Contact( "TemperatureControl".Selected )
   END_RUNG wire#w2
   RUNG wire#powerrail
      Contact( "RMAdd".Selected )
   END_RUNG wire#w2
   RUNG wire#powerrail
      Contact( "Mm01Mixing".Selected )
   END_RUNG wire#w2
   RUNG wire#powerrail
      Contact( "ProductTransfer".Selected )
   END_RUNG wire#w2
   RUNG wire#powerrail
      Contact( "BatchSAD".Fault )
   END_RUNG wire#w3
   // the same network as SCL:
   "FinalVolumeMakeup"(Enable := "ModeDb".Cycle2.Selected OR "Cycle2.Selected",   // "FB301"
                       Disable := "FinalVolumeMakeup".Running OR ("ModeDb".VesselWeight >= "FinalVolumeMakeup".FillQuantity) OR "FillWfi".Selected OR "N2Sparging".Selected OR "GasBlanketing".Selected OR "TemperatureControl".Selected OR "RMAdd".Selected OR "Mm01Mixing".Selected OR "ProductTransfer".Selected,
                       Fault := "BatchSAD".Fault,
                       SecPulse := "Sec_Pulse",
                       AlwaysTrue := "AlwaysTRUE",
                       StartConfirmationPopupSel := 0,
                       InitialDrainSel := 1,
                       FinalVolumeMakeupSel := 1,
                       UtilitySel := 1,
                       ActualQuantity := "ModeDb".VesselWeight,
                       InflightQuantity := "BatchProductionSettings".InflightQty,
                       ZDVDelay := "CommonProductionSettings".WFIDelay,
                       InitialDrainDelay := "FinalVolumeMakeup".InitialDrainDelay,
                       Start := "FinalVolumeMakeup".Start,
                       Stop := "FinalVolumeMakeup".Stop,
                       Reset := "FinalVolumeMakeup".Reset,
                       Selected := "FinalVolumeMakeup".Selected,
                       PrintTrigger => "FinalVolumeMakeup".PrintTrigger,
                       PrintWord => "FinalVolumeMakeup".PrintWord,
                       PrintStatus => "FinalVolumeMakeup".PrintStatus);
END_REGION

REGION Network 22: Final Volume Event Status
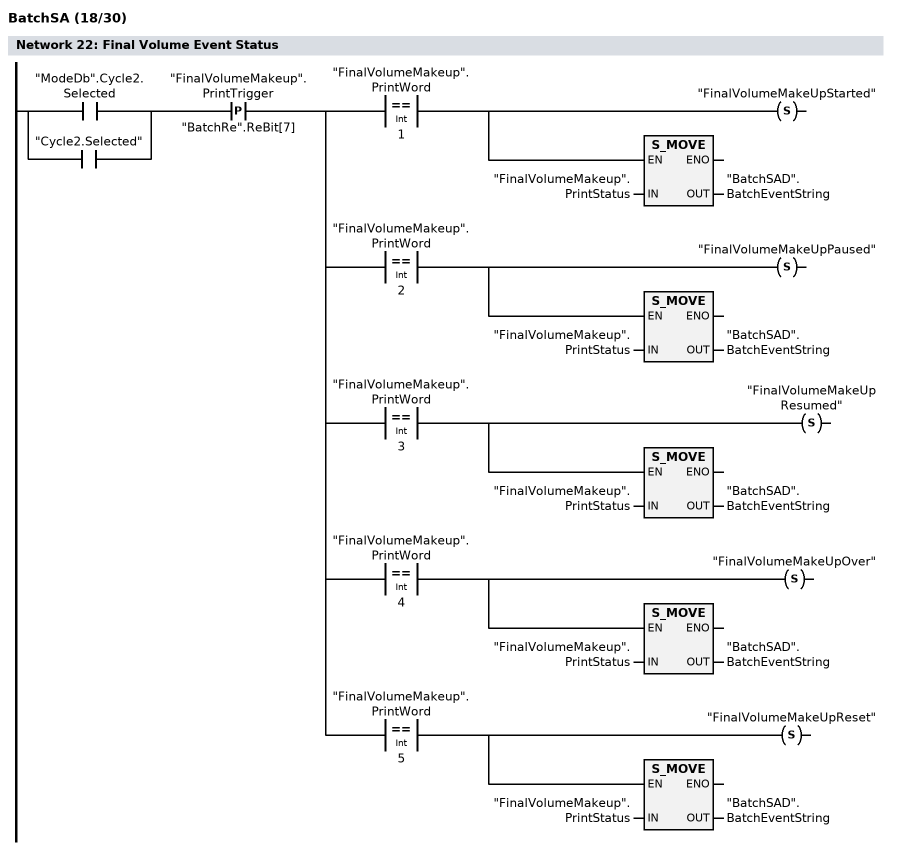
   RUNG wire#powerrail
      Contact( "ModeDb".Cycle2.Selected )
      wire#w1
      P_Contact(operand := "FinalVolumeMakeup".PrintTrigger, bit := "BatchRe".ReBit[7])
      wire#w2
      { S7_Templates := "SrcType := Int" } EQ_Contact(in1 := "FinalVolumeMakeup".PrintWord, in2 := 1)
      wire#w3
      S_Coil( "FinalVolumeMakeUpStarted" )
   END_RUNG
   RUNG wire#powerrail
      Contact( "Cycle2.Selected" )
   END_RUNG wire#w1
   RUNG wire#w3
      S_Move(in := "FinalVolumeMakeup".PrintStatus, out => "BatchSAD".BatchEventString)
   END_RUNG
   RUNG wire#w2
      { S7_Templates := "SrcType := Int" } EQ_Contact(in1 := "FinalVolumeMakeup".PrintWord, in2 := 2)
      wire#w4
      S_Coil( "FinalVolumeMakeUpPaused" )
   END_RUNG
   RUNG wire#w4
      S_Move(in := "FinalVolumeMakeup".PrintStatus, out => "BatchSAD".BatchEventString)
   END_RUNG
   RUNG wire#w2
      { S7_Templates := "SrcType := Int" } EQ_Contact(in1 := "FinalVolumeMakeup".PrintWord, in2 := 3)
      wire#w5
      S_Coil( "FinalVolumeMakeUpResumed" )
   END_RUNG
   RUNG wire#w5
      S_Move(in := "FinalVolumeMakeup".PrintStatus, out => "BatchSAD".BatchEventString)
   END_RUNG
   RUNG wire#w2
      { S7_Templates := "SrcType := Int" } EQ_Contact(in1 := "FinalVolumeMakeup".PrintWord, in2 := 4)
      wire#w6
      S_Coil( "FinalVolumeMakeUpOver" )
   END_RUNG
   RUNG wire#w6
      S_Move(in := "FinalVolumeMakeup".PrintStatus, out => "BatchSAD".BatchEventString)
   END_RUNG
   RUNG wire#w2
      { S7_Templates := "SrcType := Int" } EQ_Contact(in1 := "FinalVolumeMakeup".PrintWord, in2 := 5)
      wire#w7
      S_Coil( "FinalVolumeMakeUpReset" )
   END_RUNG
   RUNG wire#w7
      S_Move(in := "FinalVolumeMakeup".PrintStatus, out => "BatchSAD".BatchEventString)
   END_RUNG
   // the same network as SCL:
   #_w1 := ("ModeDb".Cycle2.Selected OR "Cycle2.Selected") AND "FinalVolumeMakeup".PrintTrigger AND NOT "BatchRe".ReBit[7];   // rising edge of "FinalVolumeMakeup".PrintTrigger
   "BatchRe".ReBit[7] := "FinalVolumeMakeup".PrintTrigger;
   IF #_w1 AND ("FinalVolumeMakeup".PrintWord = 1) THEN
       "FinalVolumeMakeUpStarted" := TRUE;
       "BatchSAD".BatchEventString := "FinalVolumeMakeup".PrintStatus;
   END_IF;
   IF #_w1 AND ("FinalVolumeMakeup".PrintWord = 2) THEN
       "FinalVolumeMakeUpPaused" := TRUE;
       "BatchSAD".BatchEventString := "FinalVolumeMakeup".PrintStatus;
   END_IF;
   IF #_w1 AND ("FinalVolumeMakeup".PrintWord = 3) THEN
       "FinalVolumeMakeUpResumed" := TRUE;
       "BatchSAD".BatchEventString := "FinalVolumeMakeup".PrintStatus;
   END_IF;
   IF #_w1 AND ("FinalVolumeMakeup".PrintWord = 4) THEN
       "FinalVolumeMakeUpOver" := TRUE;
       "BatchSAD".BatchEventString := "FinalVolumeMakeup".PrintStatus;
   END_IF;
   IF #_w1 AND ("FinalVolumeMakeup".PrintWord = 5) THEN
       "FinalVolumeMakeUpReset" := TRUE;
       "BatchSAD".BatchEventString := "FinalVolumeMakeup".PrintStatus;
   END_IF;
END_REGION

REGION Network 23: ******************************Product Transfer******************************
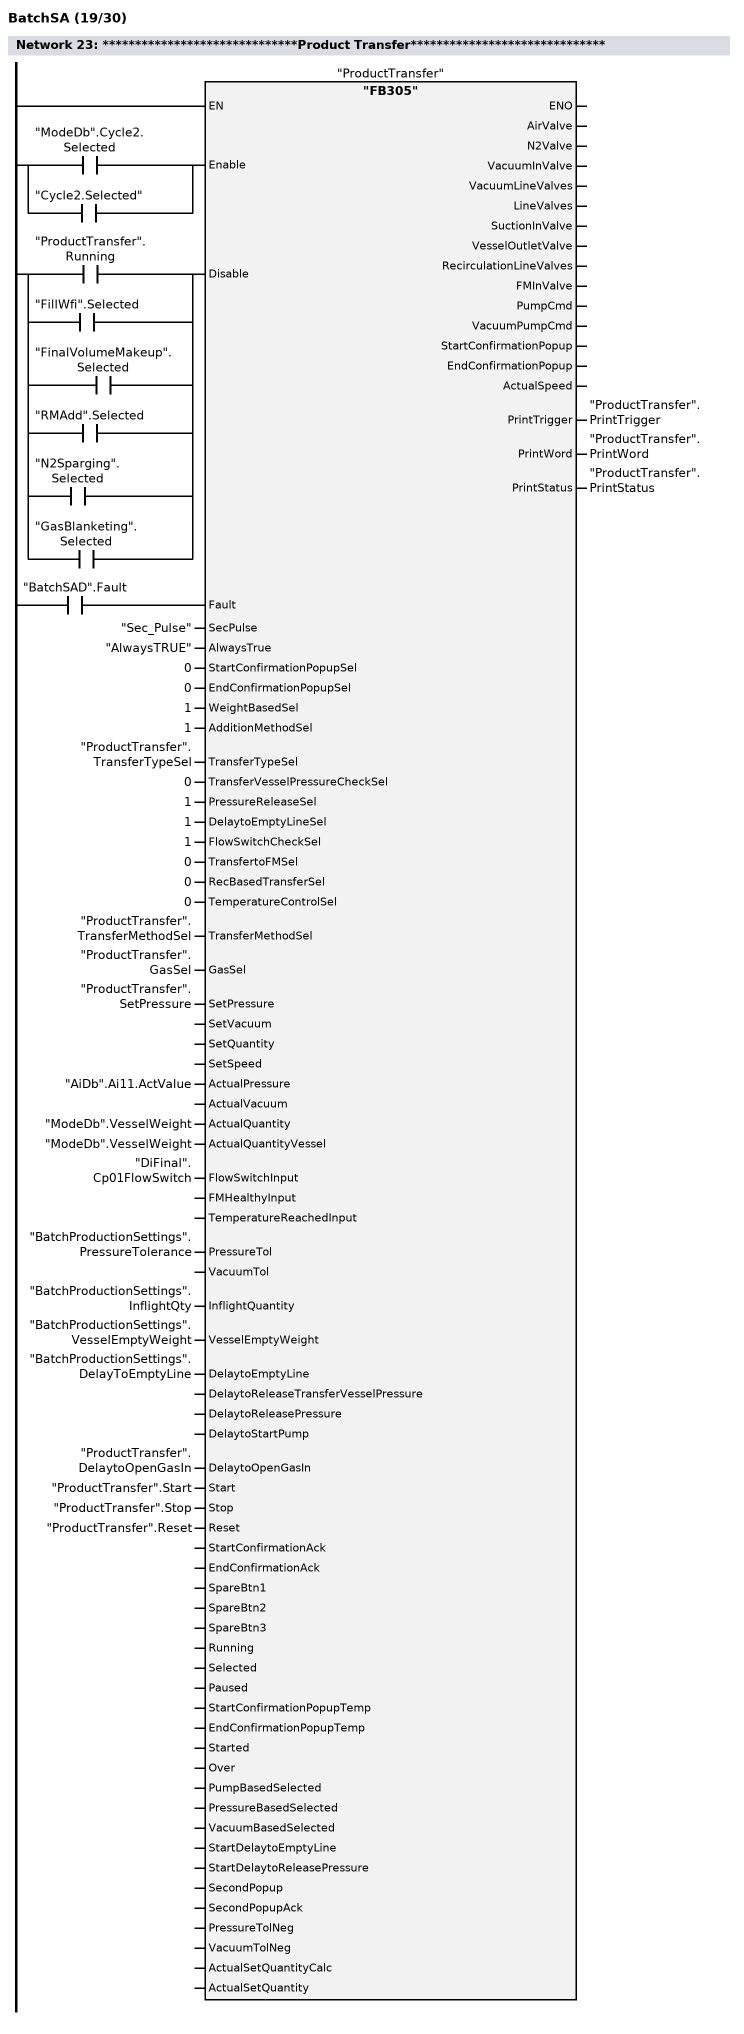
   RUNG wire#powerrail
      "ProductTransfer"(Enable := wire#w1, Disable := wire#w2, Fault := wire#w3, SecPulse := "Sec_Pulse", AlwaysTrue := "AlwaysTRUE", StartConfirmationPopupSel := 0, EndConfirmationPopupSel := 0, WeightBasedSel := 1, AdditionMethodSel := 1, TransferTypeSel := "ProductTransfer".TransferTypeSel, TransferVesselPressureCheckSel := 0, PressureReleaseSel := 1, DelaytoEmptyLineSel := 1, FlowSwitchCheckSel := 1, TransfertoFMSel := 0, RecBasedTransferSel := 0, TemperatureControlSel := 0, TransferMethodSel := "ProductTransfer".TransferMethodSel, GasSel := "ProductTransfer".GasSel, SetPressure := "ProductTransfer".SetPressure, SetVacuum :=, SetQuantity :=, SetSpeed :=, ActualPressure := "AiDb".Ai11.ActValue, ActualVacuum :=, ActualQuantity := "ModeDb".VesselWeight, ActualQuantityVessel := "ModeDb".VesselWeight, FlowSwitchInput := "DiFinal".Cp01FlowSwitch, FMHealthyInput :=, TemperatureReachedInput :=, PressureTol := "BatchProductionSettings".PressureTolerance, VacuumTol :=, InflightQuantity := "BatchProductionSettings".InflightQty, VesselEmptyWeight := "BatchProductionSettings".VesselEmptyWeight, DelaytoEmptyLine := "BatchProductionSettings".DelayToEmptyLine, DelaytoReleaseTransferVesselPressure :=, DelaytoReleasePressure :=, DelaytoStartPump :=, DelaytoOpenGasIn := "ProductTransfer".DelaytoOpenGasIn, Start := "ProductTransfer".Start, Stop := "ProductTransfer".Stop, Reset := "ProductTransfer".Reset, StartConfirmationAck :=, EndConfirmationAck :=, SpareBtn1 :=, SpareBtn2 :=, SpareBtn3 :=, Running :=, Selected :=, Paused :=, StartConfirmationPopupTemp :=, EndConfirmationPopupTemp :=, Started :=, Over :=, PumpBasedSelected :=, PressureBasedSelected :=, VacuumBasedSelected :=, StartDelaytoEmptyLine :=, StartDelaytoReleasePressure :=, SecondPopup :=, SecondPopupAck :=, PressureTolNeg :=, VacuumTolNeg :=, ActualSetQuantityCalc :=, ActualSetQuantity :=, AirValve =>, N2Valve =>, VacuumInValve =>, VacuumLineValves =>, LineValves =>, SuctionInValve =>, VesselOutletValve =>, RecirculationLineValves =>, FMInValve =>, PumpCmd =>, VacuumPumpCmd =>, StartConfirmationPopup =>, EndConfirmationPopup =>, ActualSpeed =>, PrintTrigger => "ProductTransfer".PrintTrigger, PrintWord => "ProductTransfer".PrintWord, PrintStatus => "ProductTransfer".PrintStatus)
   END_RUNG
   RUNG wire#powerrail
      Contact( "ModeDb".Cycle2.Selected )
   END_RUNG wire#w1
   RUNG wire#powerrail
      Contact( "Cycle2.Selected" )
   END_RUNG wire#w1
   RUNG wire#powerrail
      Contact( "ProductTransfer".Running )
   END_RUNG wire#w2
   RUNG wire#powerrail
      Contact( "FillWfi".Selected )
   END_RUNG wire#w2
   RUNG wire#powerrail
      Contact( "FinalVolumeMakeup".Selected )
   END_RUNG wire#w2
   RUNG wire#powerrail
      Contact( "RMAdd".Selected )
   END_RUNG wire#w2
   RUNG wire#powerrail
      Contact( "N2Sparging".Selected )
   END_RUNG wire#w2
   RUNG wire#powerrail
      Contact( "GasBlanketing".Selected )
   END_RUNG wire#w2
   RUNG wire#powerrail
      Contact( "BatchSAD".Fault )
   END_RUNG wire#w3
   // the same network as SCL:
   "ProductTransfer"(Enable := "ModeDb".Cycle2.Selected OR "Cycle2.Selected",   // "FB305"
                     Disable := "ProductTransfer".Running OR "FillWfi".Selected OR "FinalVolumeMakeup".Selected OR "RMAdd".Selected OR "N2Sparging".Selected OR "GasBlanketing".Selected,
                     Fault := "BatchSAD".Fault,
                     SecPulse := "Sec_Pulse",
                     AlwaysTrue := "AlwaysTRUE",
                     StartConfirmationPopupSel := 0,
                     EndConfirmationPopupSel := 0,
                     WeightBasedSel := 1,
                     AdditionMethodSel := 1,
                     TransferTypeSel := "ProductTransfer".TransferTypeSel,
                     TransferVesselPressureCheckSel := 0,
                     PressureReleaseSel := 1,
                     DelaytoEmptyLineSel := 1,
                     FlowSwitchCheckSel := 1,
                     TransfertoFMSel := 0,
                     RecBasedTransferSel := 0,
                     TemperatureControlSel := 0,
                     TransferMethodSel := "ProductTransfer".TransferMethodSel,
                     GasSel := "ProductTransfer".GasSel,
                     SetPressure := "ProductTransfer".SetPressure,
                     ActualPressure := "AiDb".Ai11.ActValue,
                     ActualQuantity := "ModeDb".VesselWeight,
                     ActualQuantityVessel := "ModeDb".VesselWeight,
                     FlowSwitchInput := "DiFinal".Cp01FlowSwitch,
                     PressureTol := "BatchProductionSettings".PressureTolerance,
                     InflightQuantity := "BatchProductionSettings".InflightQty,
                     VesselEmptyWeight := "BatchProductionSettings".VesselEmptyWeight,
                     DelaytoEmptyLine := "BatchProductionSettings".DelayToEmptyLine,
                     DelaytoOpenGasIn := "ProductTransfer".DelaytoOpenGasIn,
                     Start := "ProductTransfer".Start,
                     Stop := "ProductTransfer".Stop,
                     Reset := "ProductTransfer".Reset,
                     PrintTrigger => "ProductTransfer".PrintTrigger,
                     PrintWord => "ProductTransfer".PrintWord,
                     PrintStatus => "ProductTransfer".PrintStatus);
END_REGION

REGION Network 24: Delay to Open Gas
